KUKA KRL program: MyProgram_214().src

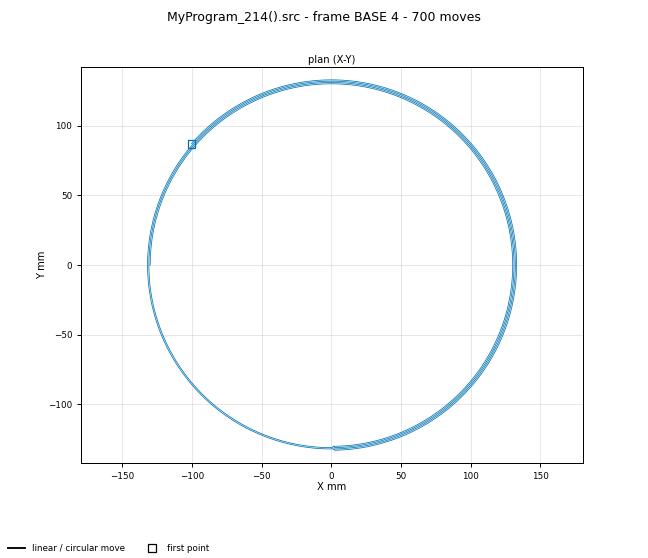
[picture p0: tool path of MyProgram_214().src in frame BASE 4, 700 of 700 moves have a stored position in this frame; points joined in program order, loops and branches not executed]
&ACCESS RVP
&REL 1
&PARAM TEMPLATE = C:\KRC\Roboter\Template\vorgabe
&PARAM EDITMASK = *
DEF MyProgram_214()
; ---- Setting reference (Base) ----
$BASE = BASE_DATA[4]

; --------------------------
; ---- Setting tool (TCP) ----
$TOOL = TOOL_DATA[3]
; --------------------------

$VEL.CP = VEL_APROX_PRINT
Startdeposition()
$VEL.CP = VEL_PRINT
LIN {X -100.4388,Y 87.0918,Z 151,A 134.8653,B 24.9546,C -1.5571,E1 24.88,E2 311.6569} C_DIS
LIN {X -97.4853,Y 90.385,Z 151,A 132.6847,B 24.9551,C -1.5488,E1 24.8842,E2 313.8668} C_DIS
LIN {X -94.8975,Y 93.098,Z 151,A 131.7947,B 24.9528,C -1.588,E1 24.8858,E2 314.6673} C_DIS
LIN {X -91.5567,Y 96.3862,Z 151,A 129.3125,B 24.9538,C -1.5705,E1 24.8908,E2 317.2017} C_DIS
LIN {X -88.2855,Y 99.3908,Z 151,A 127.4483,B 24.9534,C -1.5774,E1 24.8947,E2 319.0568} C_DIS
LIN {X -85.0766,Y 102.1512,Z 151,A 125.5893,B 24.9532,C -1.5799,E1 24.8986,E2 320.9171} C_DIS
LIN {X -81.7688,Y 104.8179,Z 151,A 123.7103,B 24.9532,C -1.5816,E1 24.9027,E2 322.799} C_DIS
LIN {X -78.285,Y 107.4446,Z 151,A 121.8187,B 24.9529,C -1.5851,E1 24.907,E2 324.689} C_DIS
LIN {X -73.7365,Y 110.6151,Z 151,A 119.6758,B 24.9519,C -1.602,E1 24.9118,E2 326.7989} C_DIS
LIN {X -71.2777,Y 112.2158,Z 151,A 117.1039,B 24.9555,C -1.5409,E1 24.9183,E2 329.5241} C_DIS
LIN {X -64.6233,Y 116.1752,Z 151,A 114.9748,B 24.9517,C -1.6057,E1 24.9231,E2 331.5056} C_DIS
LIN {X -61.5732,Y 117.8179,Z 151,A 113.4543,B 24.9517,C -1.6069,E1 24.9268,E2 333.0274} C_DIS
LIN {X -58.7566,Y 119.2473,Z 151,A 112.0651,B 24.9516,C -1.6078,E1 24.9303,E2 334.4182} C_DIS
LIN {X -55.4133,Y 120.8379,Z 151,A 110.1509,B 24.9524,C -1.5946,E1 24.9353,E2 336.3686} C_DIS
LIN {X -52.4162,Y 122.1677,Z 151,A 108.9463,B 24.9516,C -1.607,E1 24.9383,E2 337.5466} C_DIS
LIN {X -47.8757,Y 124.0173,Z 151,A 106.9413,B 24.9511,C -1.6153,E1 24.9434,E2 339.5362} C_DIS
LIN {X -44.7871,Y 125.1659,Z 151,A 105.4698,B 24.9511,C -1.6146,E1 24.9473,E2 341.0123} C_DIS
LIN {X -40.6937,Y 126.5558,Z 151,A 103.6048,B 24.9511,C -1.6168,E1 24.9522,E2 342.8756} C_DIS
LIN {X -37.2719,Y 127.6053,Z 151,A 102.1118,B 24.9508,C -1.6211,E1 24.9562,E2 344.361} C_DIS
LIN {X -33.9922,Y 128.5181,Z 151,A 100.6388,B 24.9507,C -1.6223,E1 24.9602,E2 345.8332} C_DIS
LIN {X -30.7948,Y 129.3218,Z 151,A 99.1974,B 24.9507,C -1.6227,E1 24.9641,E2 347.2758} C_DIS
LIN {X -27.1322,Y 130.1406,Z 151,A 97.4525,B 24.951,C -1.6177,E1 24.9689,E2 349.0346} C_DIS
LIN {X -23.3776,Y 130.8657,Z 151,A 95.9,B 24.9506,C -1.6239,E1 24.9731,E2 350.5742} C_DIS
LIN {X -19.5139,Y 131.4993,Z 151,A 94.2775,B 24.9503,C -1.6283,E1 24.9776,E2 352.1877} C_DIS
LIN {X -16.3255,Y 131.9325,Z 151,A 92.7599,B 24.9507,C -1.6226,E1 24.9818,E2 353.7199} C_DIS
LIN {X -12.6366,Y 132.3355,Z 151,A 91.2278,B 24.9504,C -1.6268,E1 24.986,E2 355.2429} C_DIS
LIN {X -8.7959,Y 132.6477,Z 151,A 89.4865,B 24.9506,C -1.6235,E1 24.9909,E2 356.9929} C_DIS
LIN {X -4.8875,Y 132.848,Z 151,A 87.7934,B 24.9506,C -1.6237,E1 24.9956,E2 358.6856} C_DIS
LIN {X -0.7243,Y 132.9356,Z 151,A 86.0869,B 24.9503,C -1.6287,E1 25.0004,E2 360.3806} C_DIS
LIN {X 3.3562,Y 132.8956,Z 151,A 84.2686,B 24.9505,C -1.6259,E1 25.0055,E2 362.2052} C_DIS
LIN {X 7.0592,Y 132.7505,Z 151,A 82.6113,B 24.9507,C -1.6229,E1 25.0101,E2 363.8691} C_DIS
LIN {X 11.1623,Y 132.468,Z 151,A 80.939,B 24.9503,C -1.6279,E1 25.0147,E2 365.5287} C_DIS
LIN {X 15.2217,Y 132.0641,Z 151,A 79.1094,B 24.9506,C -1.624,E1 25.0198,E2 367.3664} C_DIS
LIN {X 19.1309,Y 131.554,Z 151,A 77.4646,B 24.9504,C -1.6263,E1 25.0244,E2 369.0042} C_DIS
LIN {X 23.2351,Y 130.8912,Z 151,A 75.6881,B 24.9504,C -1.6265,E1 25.0292,E2 370.7785} C_DIS
LIN {X 26.6038,Y 130.2481,Z 151,A 74.2391,B 24.9504,C -1.6273,E1 25.0332,E2 372.2237} C_DIS
LIN {X 29.9615,Y 129.5174,Z 151,A 72.7953,B 24.9504,C -1.6285,E1 25.0371,E2 373.6629} C_DIS
LIN {X 33.2513,Y 128.7128,Z 151,A 71.0673,B 24.9512,C -1.6137,E1 25.0419,E2 375.4233} C_DIS
LIN {X 37.3957,Y 127.569,Z 151,A 69.4626,B 24.9505,C -1.6252,E1 25.0461,E2 376.9979} C_DIS
LIN {X 40.504,Y 126.6164,Z 151,A 68.0358,B 24.9507,C -1.6228,E1 25.0499,E2 378.4279} C_DIS
LIN {X 43.8865,Y 125.4846,Z 151,A 66.5342,B 24.9507,C -1.6233,E1 25.0539,E2 379.9254} C_DIS
LIN {X 47.0171,Y 124.3456,Z 151,A 65.071,B 24.9507,C -1.6205,E1 25.0577,E2 381.3922} C_DIS
LIN {X 49.9731,Y 123.187,Z 151,A 63.7361,B 24.9507,C -1.6208,E1 25.0612,E2 382.7233} C_DIS
LIN {X 53.173,Y 121.8405,Z 151,A 62.1619,B 24.9511,C -1.615,E1 25.0652,E2 384.3074} C_DIS
LIN {X 57.0541,Y 120.0715,Z 151,A 60.3594,B 24.9511,C -1.6147,E1 25.0698,E2 386.1061} C_DIS
LIN {X 60.1883,Y 118.5311,Z 151,A 58.8644,B 24.9512,C -1.6133,E1 25.0735,E2 387.6004} C_DIS
LIN {X 63.3667,Y 116.8655,Z 151,A 57.2441,B 24.9516,C -1.6072,E1 25.0776,E2 389.2304} C_DIS
LIN {X 67.1187,Y 114.7515,Z 151,A 55.3816,B 24.9518,C -1.6041,E1 25.0821,E2 391.0946} C_DIS
LIN {X 70.9545,Y 112.4198,Z 151,A 53.4788,B 24.9518,C -1.6028,E1 25.0866,E2 392.9946} C_DIS
LIN {X 74.748,Y 109.9344,Z 151,A 51.5216,B 24.9521,C -1.5994,E1 25.0911,E2 394.9532} C_DIS
LIN {X 78.4134,Y 107.351,Z 151,A 49.5804,B 24.9523,C -1.5955,E1 25.0955,E2 396.8967} C_DIS
LIN {X 81.9338,Y 104.6885,Z 151,A 47.6809,B 24.9525,C -1.5922,E1 25.0997,E2 398.7973} C_DIS
LIN {X 85.4737,Y 101.8185,Z 151,A 45.7486,B 24.9526,C -1.59,E1 25.1039,E2 400.7272} C_DIS
LIN {X 88.6689,Y 99.0484,Z 151,A 43.1234,B 24.9554,C -1.5437,E1 25.1096,E2 403.4512} C_DIS
LIN {X 93.3761,Y 94.6247,Z 151,A 41.4269,B 24.9523,C -1.5956,E1 25.1127,E2 405.0182} C_DIS
LIN {X 96.7972,Y 91.1213,Z 151,A 39.0631,B 24.9534,C -1.5773,E1 25.1174,E2 407.4151} C_DIS
LIN {X 99.9009,Y 87.7083,Z 151,A 37.0873,B 24.9536,C -1.5733,E1 25.1211,E2 409.3915} C_DIS
LIN {X 102.685,Y 84.4317,Z 151,A 34.7375,B 24.9554,C -1.5422,E1 25.1254,E2 411.8038} C_DIS
LIN {X 105.6622,Y 80.6739,Z 151,A 33.2496,B 24.9539,C -1.5681,E1 25.1278,E2 413.2235} C_DIS
LIN {X 108.0891,Y 77.392,Z 151,A 31.4386,B 24.9544,C -1.5608,E1 25.1308,E2 415.0431} C_DIS
LIN {X 111.4152,Y 72.522,Z 151,A 28.9273,B 24.9547,C -1.5558,E1 25.1347,E2 417.5538} C_DIS
LIN {X 113.7076,Y 68.8721,Z 151,A 27.0666,B 24.955,C -1.5506,E1 25.1374,E2 419.4172} C_DIS
LIN {X 115.9575,Y 65.0127,Z 151,A 25.1619,B 24.9552,C -1.5464,E1 25.14,E2 421.322} C_DIS
LIN {X 117.8536,Y 61.5051,Z 151,A 23.5076,B 24.9552,C -1.5451,E1 25.1422,E2 422.9707} C_DIS
LIN {X 119.3631,Y 58.5218,Z 151,A 22.1096,B 24.9554,C -1.5433,E1 25.1439,E2 424.3655} C_DIS
LIN {X 120.8024,Y 55.49,Z 151,A 20.682,B 24.9556,C -1.5401,E1 25.1456,E2 425.7928} C_DIS
LIN {X 122.0819,Y 52.6145,Z 151,A 19.3074,B 24.9558,C -1.5351,E1 25.1472,E2 427.1718} C_DIS
LIN {X 123.4807,Y 49.2446,Z 151,A 17.7585,B 24.956,C -1.5317,E1 25.1488,E2 428.7202} C_DIS
LIN {X 124.5747,Y 46.4055,Z 151,A 16.4792,B 24.9562,C -1.5295,E1 25.1501,E2 429.9975} C_DIS
LIN {X 125.6238,Y 43.485,Z 151,A 15.1246,B 24.9565,C -1.5245,E1 25.1513,E2 431.3563} C_DIS
LIN {X 126.7779,Y 39.9984,Z 151,A 13.4359,B 24.9571,C -1.5138,E1 25.1528,E2 433.0607} C_DIS
LIN {X 128.1939,Y 35.1996,Z 151,A 11.0831,B 24.9581,C -1.4963,E1 25.1546,E2 435.4412} C_DIS
LIN {X 129.0498,Y 31.92,Z 151,A 9.7239,B 24.9581,C -1.4972,E1 25.1555,E2 436.7903} C_DIS
LIN {X 130.1936,Y 26.8719,Z 151,A 7.6512,B 24.9579,C -1.4988,E1 25.1567,E2 438.8472} C_DIS
LIN {X 130.8791,Y 23.3024,Z 151,A 6.1872,B 24.9579,C -1.4994,E1 25.1575,E2 440.3012} C_DIS
LIN {X 131.4133,Y 20.074,Z 151,A 4.7537,B 24.9582,C -1.4936,E1 25.1581,E2 441.7401} C_DIS
LIN {X 131.9846,Y 15.8889,Z 151,A 2.9069,B 24.9586,C -1.4862,E1 25.1588,E2 443.5933} C_DIS
LIN {X 132.3916,Y 12.0521,Z 151,A 1.2035,B 24.959,C -1.4785,E1 25.1592,E2 445.3048} C_DIS
LIN {X 132.6954,Y 8.0211,Z 151,A -0.4485,B 24.959,C -1.4778,E1 25.1596,E2 446.9487} C_DIS
LIN {X 132.8828,Y 3.8181,Z 151,A -2.2288,B 24.9593,C -1.4736,E1 25.1597,E2 448.7283} C_DIS
LIN {X 132.9409,Y -0.0565,Z 151,A -4.036,B 24.96,C -1.4605,E1 25.1597,E2 450.5557} C_DIS
LIN {X 132.8768,Y -4.034,Z 151,A -5.6928,B 24.9602,C -1.458,E1 25.1597,E2 452.2084} C_DIS
LIN {X 132.6808,Y -8.2579,Z 151,A -7.4205,B 24.9602,C -1.4572,E1 25.1594,E2 453.9277} C_DIS
LIN {X 132.3492,Y -12.4942,Z 151,A -9.2116,B 24.9604,C -1.4534,E1 25.159,E2 455.7172} C_DIS
LIN {X 131.976,Y -15.9609,Z 151,A -10.686,B 24.9606,C -1.45,E1 25.1585,E2 457.191} C_DIS
LIN {X 131.4222,Y -20.0167,Z 151,A -12.4769,B 24.961,C -1.4426,E1 25.1578,E2 458.9885} C_DIS
LIN {X 130.8358,Y -23.5448,Z 151,A -13.9703,B 24.9611,C -1.4402,E1 25.1571,E2 460.4789} C_DIS
LIN {X 130.1488,Y -27.0919,Z 151,A -15.4977,B 24.9613,C -1.4367,E1 25.1563,E2 462.0056} C_DIS
LIN {X 129.5177,Y -29.9602,Z 151,A -16.8312,B 24.9618,C -1.4289,E1 25.1554,E2 463.3499} C_DIS
LIN {X 128.5065,Y -34.0359,Z 151,A -18.5829,B 24.9618,C -1.4262,E1 25.1542,E2 465.0979} C_DIS
LIN {X 127.5942,Y -37.3096,Z 151,A -20.0346,B 24.9621,C -1.4221,E1 25.1531,E2 466.5507} C_DIS
LIN {X 126.5809,Y -40.6152,Z 151,A -21.5149,B 24.9623,C -1.4179,E1 25.1519,E2 468.0327} C_DIS
LIN {X 125.5274,Y -43.7631,Z 151,A -22.9482,B 24.9626,C -1.4131,E1 25.1506,E2 469.469} C_DIS
LIN {X 124.3822,Y -46.9196,Z 151,A -24.3599,B 24.9627,C -1.4105,E1 25.1492,E2 470.8791} C_DIS
LIN {X 123.2285,Y -49.8703,Z 151,A -25.7499,B 24.963,C -1.4048,E1 25.1478,E2 472.2748} C_DIS
LIN {X 121.8935,Y -53.0503,Z 151,A -27.1857,B 24.9631,C -1.403,E1 25.1462,E2 473.707} C_DIS
LIN {X 120.6201,Y -55.8844,Z 151,A -28.5282,B 24.9634,C -1.3986,E1 25.1446,E2 475.0525} C_DIS
LIN {X 119.0684,Y -59.1193,Z 151,A -30.1178,B 24.9637,C -1.3915,E1 25.1427,E2 476.6505} C_DIS
LIN {X 116.2137,Y -64.5536,Z 151,A -32.5573,B 24.9636,C -1.3948,E1 25.1395,E2 479.0692} C_DIS
LIN {X 114.532,Y -67.4923,Z 151,A -34.2183,B 24.9644,C -1.3793,E1 25.1372,E2 480.7581} C_DIS
LIN {X 112.2366,Y -71.2448,Z 151,A -36.1169,B 24.9647,C -1.3736,E1 25.1343,E2 482.6606} C_DIS
LIN {X 109.8864,Y -74.819,Z 151,A -37.9465,B 24.9649,C -1.3691,E1 25.1315,E2 484.4918} C_DIS
LIN {X 107.4506,Y -78.2766,Z 151,A -39.7827,B 24.9652,C -1.3632,E1 25.1285,E2 486.333} C_DIS
LIN {X 104.7999,Y -81.7919,Z 151,A -41.6431,B 24.9654,C -1.36,E1 25.1254,E2 488.1922} C_DIS
LIN {X 102.1086,Y -85.128,Z 151,A -43.4777,B 24.9656,C -1.3557,E1 25.1221,E2 490.0284} C_DIS
LIN {X 99.3166,Y -88.3694,Z 151,A -45.3619,B 24.9659,C -1.3486,E1 25.1186,E2 491.9208} C_DIS
LIN {X 96.3224,Y -91.6235,Z 151,A -47.2304,B 24.9661,C -1.3458,E1 25.1151,E2 493.7879} C_DIS
LIN {X 93.3487,Y -94.6515,Z 151,A -49.085,B 24.9664,C -1.3398,E1 25.1114,E2 495.6487} C_DIS
LIN {X 90.095,Y -97.7531,Z 151,A -50.9585,B 24.9664,C -1.3386,E1 25.1076,E2 497.5174} C_DIS
LIN {X 86.8975,Y -100.6063,Z 151,A -52.82,B 24.9667,C -1.3334,E1 25.1037,E2 499.3837} C_DIS
LIN {X 83.421,Y -103.507,Z 151,A -54.7407,B 24.9668,C -1.3306,E1 25.0995,E2 501.3037} C_DIS
LIN {X 79.8391,Y -106.2948,Z 151,A -56.6606,B 24.967,C -1.3283,E1 25.0953,E2 503.222} C_DIS
LIN {X 76.3705,Y -108.8136,Z 151,A -58.5582,B 24.9673,C -1.3217,E1 25.0909,E2 505.1286} C_DIS
LIN {X 72.649,Y -111.3327,Z 151,A -60.4958,B 24.9675,C -1.3177,E1 25.0864,E2 507.0691} C_DIS
LIN {X 68.7594,Y -113.7757,Z 151,A -62.4257,B 24.9675,C -1.3166,E1 25.0819,E2 508.9956} C_DIS
LIN {X 65.1927,Y -115.8563,Z 151,A -64.1936,B 24.9677,C -1.3139,E1 25.0776,E2 510.7644} C_DIS
LIN {X 61.4606,Y -117.877,Z 151,A -65.9679,B 24.9677,C -1.3137,E1 25.0732,E2 512.5343} C_DIS
LIN {X 57.5779,Y -119.8212,Z 151,A -68.4329,B 24.9694,C -1.2789,E1 25.0668,E2 515.075} C_DIS
LIN {X 53.0533,Y -121.8922,Z 151,A -69.9699,B 24.968,C -1.3079,E1 25.0631,E2 516.5396} C_DIS
LIN {X 49.8357,Y -123.2424,Z 151,A -71.4774,B 24.968,C -1.3055,E1 25.0592,E2 518.0493} C_DIS
LIN {X 46.4907,Y -124.5428,Z 151,A -72.9745,B 24.968,C -1.306,E1 25.0553,E2 519.542} C_DIS
LIN {X 43.3991,Y -125.6536,Z 151,A -74.4019,B 24.9682,C -1.3035,E1 25.0515,E2 520.9724} C_DIS
LIN {X 40.152,Y -126.7289,Z 151,A -75.8395,B 24.9682,C -1.3037,E1 25.0477,E2 522.407} C_DIS
LIN {X 37.1235,Y -127.6487,Z 151,A -77.1963,B 24.9682,C -1.3025,E1 25.0441,E2 523.7643} C_DIS
LIN {X 34.004,Y -128.515,Z 151,A -78.6396,B 24.9684,C -1.2984,E1 25.0402,E2 525.2149} C_DIS
LIN {X 30.1478,Y -129.4749,Z 151,A -80.4613,B 24.9688,C -1.2909,E1 25.0352,E2 527.0517} C_DIS
LIN {X 25.2101,Y -130.5253,Z 151,A -82.5129,B 24.9686,C -1.2955,E1 25.0296,E2 529.0899} C_DIS
LIN {X 21.9398,Y -131.1144,Z 151,A -83.9404,B 24.9686,C -1.2946,E1 25.0257,E2 530.5179} C_DIS
LIN {X 18.1449,Y -131.6949,Z 151,A -85.7012,B 24.9689,C -1.2878,E1 25.0208,E2 532.2932} C_DIS
LIN {X 14.2924,Y -132.1669,Z 151,A -87.2717,B 24.9687,C -1.2922,E1 25.0164,E2 533.8522} C_DIS
LIN {X 10.5953,Y -132.5159,Z 151,A -88.9711,B 24.969,C -1.2862,E1 25.0117,E2 535.565} C_DIS
LIN {X 6.5449,Y -132.7764,Z 151,A -90.6231,B 24.9688,C -1.2906,E1 25.0071,E2 537.206} C_DIS
LIN {X 2.3712,Y -132.9165,Z 151,A -92.448,B 24.9688,C -1.2887,E1 25.002,E2 539.035} C_DIS
LIN {X 2.3712,Y -132.9165,Z 151,A -92.448,B 24.9688,C -1.2887,E1 25.002,E2 539.035} C_DIS
Enddeposition()
LIN {X 0.9367,Y -131.9874,Z 151,A -92.3022,B 23.9056,C -1.1253,E1 23.9322,E2 539.1469} C_DIS
Startdeposition()
$VEL.CP = VEL_PRINT
LIN {X 4.4041,Y -131.9216,Z 151,A -90.4423,B 23.9048,C -1.1435,E1 23.9375,E2 537.2427} C_DIS
LIN {X 7.9598,Y -131.7529,Z 151,A -88.9768,B 23.9049,C -1.1401,E1 23.9415,E2 535.786} C_DIS
LIN {X 11.3851,Y -131.5013,Z 151,A -87.4867,B 23.9049,C -1.1408,E1 23.9457,E2 534.2951} C_DIS
LIN {X 15.312,Y -131.1022,Z 151,A -85.8169,B 23.9049,C -1.1396,E1 23.9503,E2 532.6294} C_DIS
LIN {X 17.9111,Y -130.7743,Z 151,A -84.5466,B 23.9046,C -1.147,E1 23.9539,E2 531.3419} C_DIS
LIN {X 21.576,Y -130.2176,Z 151,A -83.0479,B 23.9048,C -1.1427,E1 23.958,E2 529.8556} C_DIS
LIN {X 25.5515,Y -129.4984,Z 151,A -81.1816,B 23.9045,C -1.1498,E1 23.9631,E2 527.9739} C_DIS
LIN {X 28.6235,Y -128.8542,Z 151,A -79.955,B 23.9047,C -1.1441,E1 23.9664,E2 526.763} C_DIS
LIN {X 32.1421,Y -128.0198,Z 151,A -78.3859,B 23.9047,C -1.1457,E1 23.9707,E2 525.1924} C_DIS
LIN {X 35.2215,Y -127.2071,Z 151,A -76.9633,B 23.9045,C -1.1492,E1 23.9746,E2 523.7636} C_DIS
LIN {X 37.9247,Y -126.4291,Z 151,A -75.6517,B 23.9042,C -1.1552,E1 23.9781,E2 522.4395} C_DIS
LIN {X 41.2838,Y -125.3711,Z 151,A -74.2316,B 23.9044,C -1.1515,E1 23.9818,E2 521.0313} C_DIS
LIN {X 44.4658,Y -124.2777,Z 151,A -72.7967,B 23.9044,C -1.1521,E1 23.9856,E2 519.5981} C_DIS
LIN {X 47.5366,Y -123.1357,Z 151,A -71.3914,B 23.9044,C -1.1532,E1 23.9893,E2 518.1933} C_DIS
LIN {X 50.5434,Y -121.9325,Z 151,A -69.9776,B 23.9042,C -1.1556,E1 23.9929,E2 516.7769} C_DIS
LIN {X 53.5713,Y -120.6328,Z 151,A -68.7335,B 23.9045,C -1.1482,E1 23.9961,E2 515.5541} C_DIS
LIN {X 56.1502,Y -119.4566,Z 151,A -67.3232,B 23.904,C -1.1594,E1 23.9997,E2 514.1202} C_DIS
LIN {X 59.5377,Y -117.8025,Z 151,A -65.8636,B 23.9043,C -1.153,E1 24.0033,E2 512.6804} C_DIS
LIN {X 62.3144,Y -116.3593,Z 151,A -64.234,B 23.9036,C -1.1693,E1 24.0074,E2 511.0154} C_DIS
LIN {X 66.1207,Y -114.2392,Z 151,A -62.3845,B 23.9036,C -1.1706,E1 24.0119,E2 509.1686} C_DIS
LIN {X 69.8904,Y -111.9728,Z 151,A -60.5105,B 23.9034,C -1.1724,E1 24.0164,E2 507.2965} C_DIS
LIN {X 73.137,Y -109.8797,Z 151,A -58.7744,B 23.9031,C -1.1788,E1 24.0204,E2 505.5505} C_DIS
LIN {X 76.7032,Y -107.4205,Z 151,A -56.9224,B 23.9031,C -1.1812,E1 24.0247,E2 503.6994} C_DIS
LIN {X 80.1465,Y -104.8765,Z 151,A -55.0654,B 23.9029,C -1.1851,E1 24.0288,E2 501.8398} C_DIS
LIN {X 83.6669,Y -102.0903,Z 151,A -53.1824,B 23.9029,C -1.186,E1 24.0329,E2 499.9621} C_DIS
LIN {X 86.9206,Y -99.3347,Z 151,A -51.3402,B 23.9026,C -1.1898,E1 24.0368,E2 498.1181} C_DIS
LIN {X 90.1019,Y -96.4584,Z 151,A -49.4852,B 23.9024,C -1.1939,E1 24.0406,E2 496.261} C_DIS
LIN {X 93.1608,Y -93.5073,Z 151,A -47.6528,B 23.9023,C -1.1977,E1 24.0443,E2 494.4272} C_DIS
LIN {X 96.1372,Y -90.4444,Z 151,A -45.7785,B 23.902,C -1.2034,E1 24.0479,E2 492.5473} C_DIS
LIN {X 99.0213,Y -87.2774,Z 151,A -43.95,B 23.9018,C -1.2066,E1 24.0513,E2 490.7195} C_DIS
LIN {X 101.7797,Y -84.0444,Z 151,A -42.1269,B 23.9017,C -1.2104,E1 24.0546,E2 488.8961} C_DIS
LIN {X 104.4375,Y -80.7179,Z 151,A -40.2901,B 23.9015,C -1.2148,E1 24.0578,E2 487.0576} C_DIS
LIN {X 106.9815,Y -77.3145,Z 151,A -38.4145,B 23.9011,C -1.2215,E1 24.0609,E2 485.1749} C_DIS
LIN {X 109.4085,Y -73.8399,Z 151,A -36.6302,B 23.9011,C -1.2238,E1 24.0637,E2 483.3942} C_DIS
LIN {X 111.5238,Y -70.6046,Z 151,A -34.8927,B 23.9006,C -1.2317,E1 24.0663,E2 481.6463} C_DIS
LIN {X 113.9272,Y -66.6573,Z 151,A -32.9195,B 23.9004,C -1.2358,E1 24.0692,E2 479.6736} C_DIS
LIN {X 116.0771,Y -62.8397,Z 151,A -31.1008,B 23.9004,C -1.2371,E1 24.0716,E2 477.8619} C_DIS
LIN {X 117.466,Y -60.1986,Z 151,A -29.8303,B 23.9002,C -1.2397,E1 24.0733,E2 476.5921} C_DIS
LIN {X 118.9463,Y -57.2182,Z 151,A -28.3968,B 23.9001,C -1.2435,E1 24.075,E2 475.1573} C_DIS
LIN {X 120.309,Y -54.2952,Z 151,A -26.9673,B 23.8998,C -1.2493,E1 24.0767,E2 473.7216} C_DIS
LIN {X 121.633,Y -51.2604,Z 151,A -25.5906,B 23.8998,C -1.2506,E1 24.0782,E2 472.3498} C_DIS
LIN {X 122.7662,Y -48.4872,Z 151,A -24.3318,B 23.8996,C -1.2524,E1 24.0795,E2 471.0938} C_DIS
LIN {X 123.8927,Y -45.5336,Z 151,A -22.7752,B 23.8989,C -1.2665,E1 24.081,E2 469.5117} C_DIS
LIN {X 125.1573,Y -41.9257,Z 151,A -21.3129,B 23.8992,C -1.2613,E1 24.0823,E2 468.0708} C_DIS
LIN {X 126.1136,Y -38.9557,Z 151,A -20.1173,B 23.8994,C -1.2572,E1 24.0833,E2 466.8925} C_DIS
LIN {X 126.9,Y -36.3195,Z 151,A -18.7563,B 23.8988,C -1.2698,E1 24.0844,E2 465.5087} C_DIS
LIN {X 127.8642,Y -32.7556,Z 151,A -17.1378,B 23.8985,C -1.2759,E1 24.0856,E2 463.8851} C_DIS
LIN {X 128.6037,Y -29.7204,Z 151,A -15.9959,B 23.8988,C -1.2689,E1 24.0863,E2 462.7673} C_DIS
LIN {X 129.2756,Y -26.6464,Z 151,A -14.469,B 23.8982,C -1.2818,E1 24.0872,E2 461.2179} C_DIS
LIN {X 129.9002,Y -23.4109,Z 151,A -13.0292,B 23.8979,C -1.287,E1 24.0879,E2 459.7743} C_DIS
LIN {X 130.4406,Y -20.1834,Z 151,A -11.6326,B 23.8977,C -1.2904,E1 24.0886,E2 458.3781} C_DIS
LIN {X 130.9162,Y -16.828,Z 151,A -10.036,B 23.8971,C -1.3018,E1 24.0892,E2 456.7632} C_DIS
LIN {X 131.3581,Y -12.9347,Z 151,A -8.4873,B 23.8973,C -1.2993,E1 24.0896,E2 455.2304} C_DIS
LIN {X 131.6194,Y -9.9294,Z 151,A -7.2018,B 23.8971,C -1.3023,E1 24.0899,E2 453.9454} C_DIS
LIN {X 131.8256,Y -6.6462,Z 151,A -5.7523,B 23.8968,C -1.3082,E1 24.0901,E2 452.4906} C_DIS
LIN {X 131.9626,Y -2.9298,Z 151,A -4.0166,B 23.8962,C -1.3199,E1 24.0903,E2 450.7371} C_DIS
LIN {X 131.987,Y 1.4617,Z 151,A -2.1672,B 23.896,C -1.3231,E1 24.0903,E2 448.8913} C_DIS
LIN {X 131.8992,Y 4.9799,Z 151,A -0.7407,B 23.896,C -1.3227,E1 24.0901,E2 447.4747} C_DIS
LIN {X 131.7237,Y 8.4341,Z 151,A 0.8861,B 23.8955,C -1.3343,E1 24.0899,E2 445.8297} C_DIS
LIN {X 131.3166,Y 13.3667,Z 151,A 2.9878,B 23.8952,C -1.3387,E1 24.0893,E2 443.7302} C_DIS
LIN {X 130.9162,Y 16.828,Z 151,A 4.3954,B 23.8952,C -1.338,E1 24.0888,E2 442.333} C_DIS
LIN {X 130.4742,Y 19.9665,Z 151,A 5.7706,B 23.895,C -1.3424,E1 24.0883,E2 440.9555} C_DIS
LIN {X 129.7915,Y 24.0182,Z 151,A 7.5045,B 23.8949,C -1.3454,E1 24.0874,E2 439.2249} C_DIS
LIN {X 129.0908,Y 27.5275,Z 151,A 9.027,B 23.8947,C -1.3488,E1 24.0866,E2 437.7036} C_DIS
LIN {X 128.5029,Y 30.1616,Z 151,A 10.3509,B 23.8941,C -1.3605,E1 24.0857,E2 436.359} C_DIS
LIN {X 127.6234,Y 33.6818,Z 151,A 11.8036,B 23.8941,C -1.3589,E1 24.0847,E2 434.9189} C_DIS
LIN {X 126.7707,Y 36.761,Z 151,A 12.9838,B 23.8945,C -1.3523,E1 24.0839,E2 433.7619} C_DIS
LIN {X 125.8816,Y 39.7003,Z 151,A 14.5027,B 23.8938,C -1.3662,E1 24.0826,E2 432.2182} C_DIS
LIN {X 124.8238,Y 42.9091,Z 151,A 15.9461,B 23.8936,C -1.3694,E1 24.0813,E2 430.7753} C_DIS
LIN {X 123.6986,Y 46.0519,Z 151,A 17.3645,B 23.8934,C -1.3722,E1 24.0799,E2 429.3585} C_DIS
LIN {X 122.5516,Y 49.0231,Z 151,A 18.7624,B 23.8932,C -1.3771,E1 24.0785,E2 427.9567} C_DIS
LIN {X 121.2821,Y 52.0844,Z 151,A 20.196,B 23.8929,C -1.3811,E1 24.077,E2 426.5216} C_DIS
LIN {X 119.9753,Y 55.0284,Z 151,A 21.5849,B 23.8928,C -1.3846,E1 24.0754,E2 425.1319} C_DIS
LIN {X 118.7411,Y 57.6478,Z 151,A 22.8341,B 23.8926,C -1.3878,E1 24.0738,E2 423.8821} C_DIS
LIN {X 117.1045,Y 60.9002,Z 151,A 24.47,B 23.8922,C -1.3952,E1 24.0718,E2 422.2371} C_DIS
LIN {X 114.9775,Y 64.8285,Z 151,A 26.428,B 23.8918,C -1.4015,E1 24.0691,E2 420.2743} C_DIS
LIN {X 112.7311,Y 68.6617,Z 151,A 28.3888,B 23.8914,C -1.4084,E1 24.0663,E2 418.3071} C_DIS
LIN {X 110.4793,Y 72.229,Z 151,A 30.1369,B 23.8914,C -1.4089,E1 24.0636,E2 416.567} C_DIS
LIN {X 108.1067,Y 75.7341,Z 151,A 32.0374,B 23.891,C -1.4169,E1 24.0606,E2 414.6566} C_DIS
LIN {X 105.4689,Y 79.3654,Z 151,A 33.9465,B 23.8908,C -1.4198,E1 24.0575,E2 412.7501} C_DIS
LIN {X 102.6282,Y 83.0061,Z 151,A 35.869,B 23.8908,C -1.4204,E1 24.0541,E2 410.8355} C_DIS
LIN {X 100.1318,Y 86.0011,Z 151,A 37.6253,B 23.8904,C -1.4277,E1 24.0509,E2 409.0696} C_DIS
LIN {X 97.2995,Y 89.1929,Z 151,A 39.4689,B 23.8901,C -1.4315,E1 24.0475,E2 407.2253} C_DIS
LIN {X 94.1083,Y 92.5537,Z 151,A 41.3987,B 23.8901,C -1.4318,E1 24.0438,E2 405.3037} C_DIS
LIN {X 91.0646,Y 95.55,Z 151,A 43.2439,B 23.8899,C -1.4353,E1 24.0401,E2 403.458} C_DIS
LIN {X 88.1979,Y 98.2023,Z 151,A 45.0036,B 23.8896,C -1.4421,E1 24.0364,E2 401.6889} C_DIS
LIN {X 84.7,Y 101.2348,Z 151,A 46.9819,B 23.8894,C -1.4444,E1 24.0322,E2 399.713} C_DIS
LIN {X 81.3895,Y 103.9149,Z 151,A 48.7723,B 23.8894,C -1.4449,E1 24.0283,E2 397.9284} C_DIS
LIN {X 77.9804,Y 106.4971,Z 151,A 50.6782,B 23.8891,C -1.4508,E1 24.024,E2 396.0152} C_DIS
LIN {X 74.3399,Y 109.0701,Z 151,A 52.6171,B 23.8889,C -1.4543,E1 24.0196,E2 394.0747} C_DIS
LIN {X 70.8092,Y 111.3947,Z 151,A 54.4709,B 23.8886,C -1.4582,E1 24.0152,E2 392.2177} C_DIS
LIN {X 67.2186,Y 113.5974,Z 151,A 56.2916,B 23.8885,C -1.4606,E1 24.0109,E2 390.397} C_DIS
LIN {X 63.3637,Y 115.7912,Z 151,A 58.1711,B 23.8885,C -1.461,E1 24.0063,E2 388.5223} C_DIS
LIN {X 60.1986,Y 117.466,Z 151,A 59.63,B 23.8886,C -1.4583,E1 24.0027,E2 387.0744} C_DIS
LIN {X 57.2182,Y 118.9463,Z 151,A 61.0822,B 23.8886,C -1.4605,E1 23.9991,E2 385.6207} C_DIS
LIN {X 54.2715,Y 120.3196,Z 151,A 62.317,B 23.8889,C -1.4533,E1 23.996,E2 384.407} C_DIS
LIN {X 51.6256,Y 121.4805,Z 151,A 63.8281,B 23.8881,C -1.4676,E1 23.992,E2 382.8644} C_DIS
LIN {X 48.5628,Y 122.7368,Z 151,A 65.2364,B 23.8881,C -1.4676,E1 23.9884,E2 381.4594} C_DIS
LIN {X 45.0038,Y 124.0837,Z 151,A 66.8008,B 23.8882,C -1.4649,E1 23.9843,E2 379.9053} C_DIS
LIN {X 42.0289,Y 125.1229,Z 151,A 68.1673,B 23.8882,C -1.466,E1 23.9807,E2 378.5389} C_DIS
LIN {X 38.9557,Y 126.1136,Z 151,A 69.5661,B 23.8882,C -1.467,E1 23.977,E2 377.1404} C_DIS
LIN {X 35.8894,Y 127.0203,Z 151,A 70.7763,B 23.8886,C -1.4591,E1 23.9738,E2 375.9516} C_DIS
LIN {X 33.2401,Y 127.7412,Z 151,A 72.2735,B 23.8877,C -1.4751,E1 23.9696,E2 374.4175} C_DIS
LIN {X 29.7204,Y 128.6037,Z 151,A 73.5313,B 23.8885,C -1.4604,E1 23.9663,E2 373.1979} C_DIS
LIN {X 26.6464,Y 129.2756,Z 151,A 75.1036,B 23.8879,C -1.4713,E1 23.962,E2 371.6008} C_DIS
LIN {X 23.6822,Y 129.8517,Z 151,A 76.4047,B 23.8879,C -1.4713,E1 23.9584,E2 370.3012} C_DIS
LIN {X 20.9589,Y 130.3205,Z 151,A 77.7047,B 23.8876,C -1.4767,E1 23.9548,E2 368.9893} C_DIS
LIN {X 17.2974,Y 130.8547,Z 151,A 79.1863,B 23.8879,C -1.471,E1 23.9507,E2 367.5231} C_DIS
LIN {X 14.198,Y 131.2271,Z 151,A 80.5251,B 23.8879,C -1.4704,E1 23.947,E2 366.1867} C_DIS
LIN {X 11.198,Y 131.5171,Z 151,A 81.7725,B 23.8881,C -1.4676,E1 23.9436,E2 364.9471} C_DIS
LIN {X 8.4341,Y 131.7237,Z 151,A 82.8678,B 23.8884,C -1.4624,E1 23.9406,E2 363.8653} C_DIS
LIN {X 5.4442,Y 131.8811,Z 151,A 84.3664,B 23.8878,C -1.4721,E1 23.9363,E2 362.3433} C_DIS
LIN {X 2.0893,Y 131.9766,Z 151,A 85.8568,B 23.8878,C -1.4735,E1 23.9321,E2 360.8494} C_DIS
LIN {X -2.0372,Y 131.9775,Z 151,A 87.538,B 23.8881,C -1.4678,E1 23.9275,E2 359.1824} C_DIS
LIN {X -4.9465,Y 131.9005,Z 151,A 88.8969,B 23.8878,C -1.4721,E1 23.9237,E2 357.8127} C_DIS
LIN {X -8.4341,Y 131.7237,Z 151,A 90.5328,B 23.8875,C -1.4774,E1 23.9191,E2 356.1633} C_DIS
LIN {X -12.3279,Y 131.4163,Z 151,A 92.054,B 23.8881,C -1.4681,E1 23.9149,E2 354.6641} C_DIS
LIN {X -15.312,Y 131.1022,Z 151,A 93.3721,B 23.8881,C -1.4681,E1 23.9112,E2 353.3451} C_DIS
LIN {X -17.9111,Y 130.7743,Z 151,A 94.6462,B 23.8877,C -1.474,E1 23.9077,E2 352.0554} C_DIS
LIN {X -20.9589,Y 130.3205,Z 151,A 95.9891,B 23.8877,C -1.4734,E1 23.904,E2 350.713} C_DIS
LIN {X -24.0182,Y 129.7915,Z 151,A 97.3655,B 23.8877,C -1.4737,E1 23.9002,E2 349.3341} C_DIS
LIN {X -27.5275,Y 129.0908,Z 151,A 98.5901,B 23.8887,C -1.4566,E1 23.8969,E2 348.1504} C_DIS
LIN {X -30.1616,Y 128.5029,Z 151,A 100.0787,B 23.8879,C -1.4707,E1 23.8928,E2 346.6248} C_DIS
LIN {X -33.6818,Y 127.6234,Z 151,A 101.5224,B 23.8884,C -1.4629,E1 23.8889,E2 345.1983} C_DIS
LIN {X -36.9312,Y 126.7209,Z 151,A 102.9932,B 23.8884,C -1.4617,E1 23.885,E2 343.728} C_DIS
LIN {X -40.9339,Y 125.4876,Z 151,A 104.9571,B 23.8882,C -1.4665,E1 23.8797,E2 341.7485} C_DIS
LIN {X -44.4417,Y 124.2864,Z 151,A 106.4566,B 23.8886,C -1.4592,E1 23.8758,E2 340.2638} C_DIS
LIN {X -47.5765,Y 123.1202,Z 151,A 107.8995,B 23.8887,C -1.4569,E1 23.872,E2 338.8236} C_DIS
LIN {X -50.5434,Y 121.9325,Z 151,A 109.2839,B 23.8888,C -1.4548,E1 23.8685,E2 337.4412} C_DIS
LIN {X -53.5713,Y 120.6328,Z 151,A 110.5358,B 23.8894,C -1.4442,E1 23.8653,E2 336.2123} C_DIS
LIN {X -56.1502,Y 119.4566,Z 151,A 111.9562,B 23.889,C -1.4513,E1 23.8617,E2 334.7707} C_DIS
LIN {X -59.4899,Y 117.8268,Z 151,A 113.5879,B 23.8891,C -1.4496,E1 23.8576,E2 333.1387} C_DIS
LIN {X -62.8397,Y 116.0771,Z 151,A 115.3531,B 23.8889,C -1.4527,E1 23.8532,E2 331.3606} C_DIS
LIN {X -66.7018,Y 113.901,Z 151,A 117.2623,B 23.8892,C -1.4485,E1 23.8486,E2 329.4557} C_DIS
LIN {X -70.6046,Y 111.5238,Z 151,A 119.2153,B 23.8895,C -1.4434,E1 23.844,E2 327.5092} C_DIS
LIN {X -73.8399,Y 109.4085,Z 151,A 120.9426,B 23.8895,C -1.4424,E1 23.8399,E2 325.7782} C_DIS
LIN {X -77.3145,Y 106.9815,Z 151,A 122.7919,B 23.8897,C -1.4391,E1 23.8357,E2 323.9305} C_DIS
LIN {X -80.9409,Y 104.2646,Z 151,A 124.7196,B 23.8901,C -1.4331,E1 23.8315,E2 322.0103} C_DIS
LIN {X -84.0444,Y 101.7797,Z 151,A 126.5042,B 23.8901,C -1.432,E1 23.8276,E2 320.2213} C_DIS
LIN {X -87.561,Y 98.7706,Z 151,A 128.4508,B 23.8905,C -1.4245,E1 23.8235,E2 318.2853} C_DIS
LIN {X -90.6029,Y 95.9877,Z 151,A 130.2981,B 23.8906,C -1.423,E1 23.8197,E2 316.4338} C_DIS
LIN {X -93.5073,Y 93.1608,Z 151,A 132.0921,B 23.8908,C -1.4203,E1 23.8162,E2 314.6386} C_DIS
LIN {X -96.7204,Y 89.8205,Z 151,A 134.0419,B 23.8912,C -1.4124,E1 23.8125,E2 312.6994} C_DIS
LIN {X -99.4098,Y 86.8345,Z 151,A 135.8436,B 23.8913,C -1.4106,E1 23.8091,E2 310.8938} C_DIS
LIN {X -102.0903,Y 83.6669,Z 151,A 137.6801,B 23.8915,C -1.4075,E1 23.8058,E2 309.0561} C_DIS
LIN {X -104.9555,Y 80.0432,Z 151,A 139.6237,B 23.892,C -1.3992,E1 23.8025,E2 307.1233} C_DIS
LIN {X -107.4945,Y 76.5996,Z 151,A 141.4861,B 23.8922,C -1.3943,E1 23.7995,E2 305.2634} C_DIS
LIN {X -109.8797,Y 73.137,Z 151,A 143.3266,B 23.8925,C -1.3899,E1 23.7966,E2 303.4243} C_DIS
LIN {X -112.1812,Y 69.5555,Z 151,A 145.2413,B 23.8925,C -1.3877,E1 23.7937,E2 301.5049} C_DIS
LIN {X -114.4439,Y 65.767,Z 151,A 147.2081,B 23.8928,C -1.3845,E1 23.7909,E2 299.5354} C_DIS
LIN {X -116.4728,Y 62.1031,Z 151,A 149.0526,B 23.893,C -1.3803,E1 23.7885,E2 297.691} C_DIS
LIN {X -118.2163,Y 58.7116,Z 151,A 150.5725,B 23.8936,C -1.3692,E1 23.7866,E2 296.1902} C_DIS
LIN {X -119.6559,Y 55.719,Z 151,A 151.8375,B 23.8943,C -1.3567,E1 23.7851,E2 294.9489} C_DIS
LIN {X -120.8263,Y 53.1387,Z 151,A 153.3899,B 23.8937,C -1.3677,E1 23.7833,E2 293.3602} C_DIS
LIN {X -122.1605,Y 49.9935,Z 151,A 154.8467,B 23.894,C -1.3619,E1 23.7818,E2 291.9093} C_DIS
LIN {X -123.529,Y 46.5045,Z 151,A 156.31,B 23.8947,C -1.3494,E1 23.7803,E2 290.4685} C_DIS
LIN {X -124.5882,Y 43.5887,Z 151,A 157.7668,B 23.8947,C -1.3502,E1 23.7789,E2 289.001} C_DIS
LIN {X -125.6785,Y 40.3361,Z 151,A 159.195,B 23.895,C -1.3427,E1 23.7777,E2 287.5828} C_DIS
LIN {X -126.6117,Y 37.3042,Z 151,A 160.5608,B 23.8953,C -1.3378,E1 23.7766,E2 286.2209} C_DIS
LIN {X -127.3306,Y 34.7799,Z 151,A 161.7699,B 23.8953,C -1.3373,E1 23.7757,E2 285.0056} C_DIS
LIN {X -128.251,Y 31.2067,Z 151,A 163.415,B 23.8955,C -1.3342,E1 23.7746,E2 283.3582} C_DIS
LIN {X -129.2756,Y 26.6464,Z 151,A 165.4206,B 23.8959,C -1.3266,E1 23.7734,E2 281.3591} C_DIS
LIN {X -129.7915,Y 24.0182,Z 151,A 166.7247,B 23.8957,C -1.3292,E1 23.7727,E2 280.0402} C_DIS
LIN {X -130.3205,Y 20.9589,Z 151,A 168.1118,B 23.8959,C -1.3266,E1 23.7721,E2 278.6509} C_DIS
LIN {X -130.7743,Y 17.9111,Z 151,A 169.2904,B 23.8965,C -1.315,E1 23.7716,E2 277.4938} C_DIS
LIN {X -131.2006,Y 14.4442,Z 151,A 170.8589,B 23.8965,C -1.3125,E1 23.7711,E2 275.9218} C_DIS
LIN {X -131.4733,Y 11.7171,Z 151,A 172.0957,B 23.8967,C -1.3107,E1 23.7708,E2 274.6815} C_DIS
LIN {X -131.7237,Y 8.4341,Z 151,A 173.2812,B 23.8975,C -1.2949,E1 23.7706,E2 273.5278} C_DIS
LIN {X -131.8857,Y 5.3247,Z 151,A 174.6055,B 23.8978,C -1.2892,E1 23.7704,E2 272.2091} C_DIS
LIN {X -131.9696,Y 2.5087,Z 151,A 175.8718,B 23.8978,C -1.2872,E1 23.7704,E2 270.9399} C_DIS
LIN {X -131.9946,Y -0.3989,Z 151,A 177.2332,B 23.8978,C -1.2876,E1 23.7703,E2 269.5689} C_DIS
LIN {X -131.9509,Y -3.3526,Z 151,A 178.4354,B 23.8983,C -1.2798,E1 23.7703,E2 268.3785} C_DIS
LIN {X -131.8364,Y -6.4304,Z 151,A 179.9922,B 23.898,C -1.2855,E1 23.7705,E2 266.7976} C_DIS
LIN {X -131.5517,Y -10.7894,Z 151,A -178.3052,B 23.8987,C -1.2705,E1 23.7709,E2 265.1216} C_DIS
LIN {X -131.2545,Y -13.944,Z 151,A -176.7867,B 23.8987,C -1.2726,E1 23.7713,E2 263.5882} C_DIS
LIN {X -130.9162,Y -16.828,Z 151,A -175.4398,B 23.8987,C -1.2725,E1 23.7717,E2 262.2331} C_DIS
LIN {X -130.489,Y -19.8709,Z 151,A -174.2483,B 23.8992,C -1.2617,E1 23.7722,E2 261.061} C_DIS
LIN {X -129.9869,Y -22.9264,Z 151,A -172.9495,B 23.8995,C -1.2553,E1 23.7728,E2 259.7698} C_DIS
LIN {X -129.4984,Y -25.5515,Z 151,A -171.4571,B 23.8989,C -1.267,E1 23.7736,E2 258.2393} C_DIS
LIN {X -128.7326,Y -29.1557,Z 151,A -169.9683,B 23.8994,C -1.2569,E1 23.7745,E2 256.7664} C_DIS
LIN {X -127.9835,Y -32.2854,Z 151,A -168.6052,B 23.8997,C -1.251,E1 23.7754,E2 255.4096} C_DIS
LIN {X -127.2071,Y -35.2215,Z 151,A -167.2149,B 23.8997,C -1.2502,E1 23.7764,E2 254.0127} C_DIS
LIN {X -126.3202,Y -38.2807,Z 151,A -165.8901,B 23.9001,C -1.2433,E1 23.7775,E2 252.6971} C_DIS
LIN {X -125.3122,Y -41.4604,Z 151,A -164.4257,B 23.9002,C -1.2396,E1 23.7787,E2 251.2329} C_DIS
LIN {X -124.2864,Y -44.4417,Z 151,A -163.0216,B 23.9004,C -1.2372,E1 23.78,E2 249.8266} C_DIS
LIN {X -123.1503,Y -47.4991,Z 151,A -161.5946,B 23.9005,C -1.2335,E1 23.7814,E2 248.4003} C_DIS
LIN {X -121.9325,Y -50.5434,Z 151,A -160.137,B 23.9007,C -1.2309,E1 23.783,E2 246.9406} C_DIS
LIN {X -120.6328,Y -53.5713,Z 151,A -158.9045,B 23.9013,C -1.2175,E1 23.7843,E2 245.734} C_DIS
LIN {X -119.2834,Y -56.5127,Z 151,A -157.3116,B 23.9011,C -1.2222,E1 23.7862,E2 244.1203} C_DIS
LIN {X -117.8832,Y -59.3792,Z 151,A -155.8325,B 23.9011,C -1.2227,E1 23.7881,E2 242.6317} C_DIS
LIN {X -116.0771,Y -62.8397,Z 151,A -154.0746,B 23.9011,C -1.2209,E1 23.7904,E2 240.8685} C_DIS
LIN {X -113.901,Y -66.7018,Z 151,A -152.1615,B 23.9014,C -1.2151,E1 23.7931,E2 238.9591} C_DIS
LIN {X -111.5238,Y -70.6046,Z 151,A -150.2368,B 23.9018,C -1.2071,E1 23.7959,E2 237.044} C_DIS
LIN {X -109.2519,Y -74.0714,Z 151,A -148.4116,B 23.902,C -1.2036,E1 23.7987,E2 235.2179} C_DIS
LIN {X -106.8921,Y -77.4378,Z 151,A -146.591,B 23.9021,C -1.2008,E1 23.8017,E2 233.395} C_DIS
LIN {X -104.3871,Y -80.7828,Z 151,A -144.743,B 23.9023,C -1.1979,E1 23.8048,E2 231.5448} C_DIS
LIN {X -101.5443,Y -84.3287,Z 151,A -142.7893,B 23.9025,C -1.1923,E1 23.8082,E2 229.5955} C_DIS
LIN {X -98.7387,Y -87.5972,Z 151,A -140.8869,B 23.9026,C -1.1895,E1 23.8117,E2 227.691} C_DIS
LIN {X -95.7193,Y -90.8875,Z 151,A -138.8953,B 23.9027,C -1.1877,E1 23.8155,E2 225.6948} C_DIS
LIN {X -92.7286,Y -93.9368,Z 151,A -137.0317,B 23.9029,C -1.1841,E1 23.8192,E2 223.8317} C_DIS
LIN {X -89.6412,Y -96.8874,Z 151,A -135.1714,B 23.9031,C -1.1806,E1 23.823,E2 221.9722} C_DIS
LIN {X -86.3776,Y -99.8075,Z 151,A -133.2671,B 23.9032,C -1.177,E1 23.827,E2 220.0689} C_DIS
LIN {X -83.0061,Y -102.6282,Z 151,A -131.3708,B 23.9034,C -1.1728,E1 23.8311,E2 218.1755} C_DIS
LIN {X -79.3654,Y -105.4689,Z 151,A -129.4319,B 23.9037,C -1.166,E1 23.8354,E2 216.246} C_DIS
LIN {X -76.2283,Y -107.7581,Z 151,A -127.6681,B 23.9037,C -1.1668,E1 23.8394,E2 214.4737} C_DIS
LIN {X -72.4212,Y -110.3528,Z 151,A -125.6748,B 23.9039,C -1.1632,E1 23.844,E2 212.4824} C_DIS
LIN {X -68.6617,Y -112.7311,Z 151,A -123.7018,B 23.9039,C -1.1623,E1 23.8487,E2 210.5051} C_DIS
LIN {X -64.8285,Y -114.9775,Z 151,A -121.7935,B 23.9041,C -1.1585,E1 23.8533,E2 208.6003} C_DIS
LIN {X -61.6791,Y -116.6955,Z 151,A -120.3366,B 23.9044,C -1.1516,E1 23.8569,E2 207.1562} C_DIS
LIN {X -58.6088,Y -118.267,Z 151,A -118.8672,B 23.9045,C -1.1484,E1 23.8605,E2 205.6907} C_DIS
LIN {X -55.719,Y -119.6559,Z 151,A -117.6261,B 23.9049,C -1.1394,E1 23.8636,E2 204.4685} C_DIS
LIN {X -52.9089,Y -120.9256,Z 151,A -116.1228,B 23.9047,C -1.1458,E1 23.8675,E2 202.9453} C_DIS
LIN {X -49.6003,Y -122.3189,Z 151,A -114.575,B 23.9047,C -1.1437,E1 23.8715,E2 201.3991} C_DIS
LIN {X -46.6985,Y -123.4564,Z 151,A -113.2254,B 23.9048,C -1.1422,E1 23.875,E2 200.0502} C_DIS
LIN {X -43.4608,Y -124.6326,Z 151,A -111.7201,B 23.9048,C -1.1414,E1 23.8789,E2 198.5439} C_DIS
LIN {X -40.4752,Y -125.6341,Z 151,A -110.3288,B 23.9048,C -1.1414,E1 23.8826,E2 197.1497} C_DIS
LIN {X -37.8587,Y -126.4493,Z 151,A -109.1329,B 23.9048,C -1.1409,E1 23.8858,E2 195.9531} C_DIS
LIN {X -34.7799,Y -127.3306,Z 151,A -107.743,B 23.9049,C -1.1399,E1 23.8896,E2 194.5632} C_DIS
LIN {X -31.2591,Y -128.2383,Z 151,A -106.1655,B 23.9049,C -1.139,E1 23.8938,E2 192.9857} C_DIS
LIN {X -28.018,Y -128.9849,Z 151,A -104.7543,B 23.9051,C -1.1367,E1 23.8977,E2 191.5783} C_DIS
LIN {X -25.1117,Y -129.5825,Z 151,A -103.6077,B 23.9054,C -1.1292,E1 23.9008,E2 190.4489} C_DIS
LIN {X -22.0489,Y -130.1387,Z 151,A -102.0568,B 23.905,C -1.1386,E1 23.9051,E2 188.8732} C_DIS
LIN {X -18.7388,Y -130.656,Z 151,A -100.6082,B 23.905,C -1.1379,E1 23.9091,E2 187.4249} C_DIS
LIN {X -15.312,Y -131.1022,Z 151,A -99.0391,B 23.9049,C -1.1411,E1 23.9135,E2 185.8469} C_DIS
LIN {X -11.8603,Y -131.4612,Z 151,A -97.5007,B 23.9049,C -1.1425,E1 23.9178,E2 184.3041} C_DIS
LIN {X -8.4341,Y -131.7237,Z 151,A -96.0838,B 23.9049,C -1.1388,E1 23.9217,E2 182.8958} C_DIS
LIN {X -4.9783,Y -131.8992,Z 151,A -94.5713,B 23.9049,C -1.1394,E1 23.9259,E2 181.3814} C_DIS
LIN {X 0,Y -131.9951,Z 151,A -92.3458,B 23.9048,C -1.143,E1 23.9322,E2 179.1469} C_DIS
LIN {X 0,Y -131.9951,Z 151,A -92.3458,B 23.9048,C -1.143,E1 23.9322,E2 179.1469} C_DIS
Enddeposition()
LIN {X 0.9375,Y -131.0445,Z 151,A -92.4391,B 22.8257,C -0.9274,E1 22.8438,E2 179.6503} C_DIS
Startdeposition()
$VEL.CP = VEL_PRINT
LIN {X -3.5036,Y -131.0018,Z 151,A -94.3186,B 22.8257,C -0.93,E1 22.8385,E2 181.5233} C_DIS
LIN {X -7.4624,Y -130.8372,Z 151,A -95.935,B 22.8254,C -0.9353,E1 22.8341,E2 183.1265} C_DIS
LIN {X -10.4413,Y -130.6332,Z 151,A -97.2575,B 22.8254,C -0.9345,E1 22.8304,E2 184.4515} C_DIS
LIN {X -14.0931,Y -130.2885,Z 151,A -98.9617,B 22.8256,C -0.93,E1 22.8256,E2 186.1684} C_DIS
LIN {X -18.1392,Y -129.7876,Z 151,A -100.7482,B 22.8256,C -0.9302,E1 22.8207,E2 187.9558} C_DIS
LIN {X -21.576,Y -129.26,Z 151,A -102.1378,B 22.8253,C -0.9367,E1 22.8169,E2 189.3301} C_DIS
LIN {X -23.9998,Y -128.8334,Z 151,A -103.6,B 22.826,C -0.9193,E1 22.8127,E2 190.8389} C_DIS
LIN {X -28.9062,Y -127.8208,Z 151,A -105.5176,B 22.8255,C -0.9329,E1 22.8076,E2 192.724} C_DIS
LIN {X -33.4186,Y -126.7161,Z 151,A -107.5572,B 22.8255,C -0.9336,E1 22.8021,E2 194.7648} C_DIS
LIN {X -36.2814,Y -125.927,Z 151,A -108.9292,B 22.8255,C -0.9311,E1 22.7983,E2 196.1457} C_DIS
LIN {X -39.7283,Y -124.8812,Z 151,A -110.4216,B 22.8254,C -0.9361,E1 22.7944,E2 197.6281} C_DIS
LIN {X -42.9463,Y -123.8113,Z 151,A -111.9131,B 22.8254,C -0.9369,E1 22.7904,E2 199.1206} C_DIS
LIN {X -46.0619,Y -122.6863,Z 151,A -113.3861,B 22.8254,C -0.9371,E1 22.7866,E2 200.5964} C_DIS
LIN {X -49.4737,Y -121.3516,Z 151,A -115.1031,B 22.8254,C -0.9335,E1 22.7821,E2 202.327} C_DIS
LIN {X -53.0301,Y -119.8402,Z 151,A -116.6494,B 22.8251,C -0.9418,E1 22.7782,E2 203.8558} C_DIS
LIN {X -56.4823,Y -118.2512,Z 151,A -118.3197,B 22.8251,C -0.9434,E1 22.7739,E2 205.5267} C_DIS
LIN {X -59.506,Y -116.7588,Z 151,A -119.9391,B 22.8253,C -0.9387,E1 22.7699,E2 207.1629} C_DIS
LIN {X -64.4518,Y -114.1058,Z 151,A -122.3812,B 22.8251,C -0.9426,E1 22.7639,E2 209.6028} C_DIS
LIN {X -68.2431,Y -111.8798,Z 151,A -124.316,B 22.8251,C -0.9448,E1 22.7592,E2 211.5382} C_DIS
LIN {X -70.6468,Y -110.3772,Z 151,A -125.7172,B 22.8252,C -0.9396,E1 22.7559,E2 212.9581} C_DIS
LIN {X -74.3819,Y -107.8958,Z 151,A -128.0918,B 22.8258,C -0.9245,E1 22.7503,E2 215.3806} C_DIS
LIN {X -78.5841,Y -104.8751,Z 151,A -129.8145,B 22.8247,C -0.9523,E1 22.7466,E2 217.0381} C_DIS
LIN {X -82.1254,Y -102.1251,Z 151,A -131.7497,B 22.8245,C -0.957,E1 22.7424,E2 218.9691} C_DIS
LIN {X -85.5404,Y -99.2821,Z 151,A -133.6798,B 22.8244,C -0.9613,E1 22.7383,E2 220.8963} C_DIS
LIN {X -88.8911,Y -96.294,Z 151,A -135.396,B 22.8238,C -0.9761,E1 22.7348,E2 222.5817} C_DIS
LIN {X -91.3262,Y -93.9876,Z 151,A -137.0751,B 22.824,C -0.9698,E1 22.7313,E2 224.2849} C_DIS
LIN {X -94.2769,Y -91.0274,Z 151,A -138.9538,B 22.824,C -0.9715,E1 22.7276,E2 226.1681} C_DIS
LIN {X -97.3277,Y -87.7586,Z 151,A -140.9989,B 22.824,C -0.9719,E1 22.7238,E2 228.2222} C_DIS
LIN {X -100.3117,Y -84.3307,Z 151,A -142.9491,B 22.8237,C -0.9781,E1 22.7202,E2 230.166} C_DIS
LIN {X -103.2115,Y -80.756,Z 151,A -144.9405,B 22.8235,C -0.9838,E1 22.7168,E2 232.1529} C_DIS
LIN {X -105.8,Y -77.334,Z 151,A -146.8398,B 22.8233,C -0.9875,E1 22.7136,E2 234.0529} C_DIS
LIN {X -108.221,Y -73.9081,Z 151,A -148.6884,B 22.8232,C -0.9915,E1 22.7107,E2 235.9012} C_DIS
LIN {X -110.07,Y -71.125,Z 151,A -150.3855,B 22.8234,C -0.985,E1 22.708,E2 237.6245} C_DIS
LIN {X -111.8098,Y -68.3571,Z 151,A -152.7849,B 22.8249,C -0.9474,E1 22.7045,E2 240.1351} C_DIS
LIN {X -115.825,Y -61.3053,Z 151,A -155.1088,B 22.8224,C -1.0094,E1 22.7015,E2 242.3119} C_DIS
LIN {X -117.4387,Y -58.153,Z 151,A -156.6354,B 22.8222,C -1.0147,E1 22.6996,E2 243.834} C_DIS
LIN {X -118.8163,Y -55.2844,Z 151,A -158.1139,B 22.8222,C -1.0148,E1 22.6978,E2 245.3209} C_DIS
LIN {X -120.3058,Y -51.9625,Z 151,A -159.5032,B 22.8216,C -1.0281,E1 22.6963,E2 246.6841} C_DIS
LIN {X -121.9487,Y -47.9833,Z 151,A -161.5885,B 22.8218,C -1.0249,E1 22.6941,E2 248.7908} C_DIS
LIN {X -123.1613,Y -44.7776,Z 151,A -162.8606,B 22.8212,C -1.039,E1 22.6929,E2 250.0341} C_DIS
LIN {X -124.4475,Y -41.0679,Z 151,A -164.8732,B 22.8215,C -1.0314,E1 22.691,E2 252.0792} C_DIS
LIN {X -125.6973,Y -37.066,Z 151,A -166.6256,B 22.8211,C -1.0404,E1 22.6896,E2 253.8194} C_DIS
LIN {X -126.5952,Y -33.8717,Z 151,A -168.058,B 22.8209,C -1.0457,E1 22.6886,E2 255.2474} C_DIS
LIN {X -127.3942,Y -30.7306,Z 151,A -169.5276,B 22.8208,C -1.0478,E1 22.6876,E2 256.721} C_DIS
LIN {X -128.2558,Y -26.9196,Z 151,A -171.3284,B 22.8208,C -1.0491,E1 22.6865,E2 258.5301} C_DIS
LIN {X -129.0137,Y -23.0031,Z 151,A -173.0412,B 22.8204,C -1.056,E1 22.6856,E2 260.2364} C_DIS
LIN {X -129.7044,Y -18.7209,Z 151,A -175.4155,B 22.821,C -1.0417,E1 22.6846,E2 262.6635} C_DIS
LIN {X -130.2548,Y -14.4057,Z 151,A -177.5964,B 22.8213,C -1.036,E1 22.684,E2 264.8736} C_DIS
LIN {X -130.7603,Y -8.7121,Z 151,A -179.2562,B 22.8194,C -1.0794,E1 22.6836,E2 266.4316} C_DIS
LIN {X -131.0433,Y -1.3504,Z 151,A 176.5083,B 22.8208,C -1.047,E1 22.6833,E2 270.7797} C_DIS
LIN {X -130.9565,Y 4.9154,Z 151,A 174.9203,B 22.8182,C -1.1045,E1 22.6835,E2 272.229} C_DIS
LIN {X -130.521,Y 11.7691,Z 151,A 170.754,B 22.82,C -1.0649,E1 22.6844,E2 276.5257} C_DIS
LIN {X -129.8245,Y 17.8811,Z 151,A 168.8299,B 22.8182,C -1.1058,E1 22.685,E2 278.3565} C_DIS
LIN {X -129.2356,Y 21.7221,Z 151,A 166.2893,B 22.8195,C -1.0759,E1 22.6863,E2 280.9914} C_DIS
LIN {X -128.0202,Y 28.011,Z 151,A 164.2579,B 22.8177,C -1.1171,E1 22.6874,E2 282.9291} C_DIS
LIN {X -127.087,Y 31.9784,Z 151,A 162.7207,B 22.8169,C -1.1332,E1 22.6883,E2 284.4345} C_DIS
LIN {X -125.9739,Y 36.1213,Z 151,A 160.6004,B 22.8171,C -1.1287,E1 22.6899,E2 286.5802} C_DIS
LIN {X -124.9043,Y 39.6559,Z 151,A 159.0655,B 22.8167,C -1.1372,E1 22.6912,E2 288.1028} C_DIS
LIN {X -123.7815,Y 43.0322,Z 151,A 157.4977,B 22.8165,C -1.1415,E1 22.6926,E2 289.6693} C_DIS
LIN {X -122.4594,Y 46.6675,Z 151,A 155.8197,B 22.8162,C -1.1472,E1 22.6942,E2 291.3428} C_DIS
LIN {X -121.0763,Y 50.1425,Z 151,A 154.1246,B 22.8162,C -1.1497,E1 22.696,E2 293.042} C_DIS
LIN {X -119.3916,Y 54.033,Z 151,A 152.0332,B 22.8163,C -1.1452,E1 22.6984,E2 295.1579} C_DIS
LIN {X -117.332,Y 58.3694,Z 151,A 150.0407,B 22.8158,C -1.156,E1 22.7008,E2 297.1343} C_DIS
LIN {X -115.2282,Y 62.4236,Z 151,A 148.0348,B 22.8156,C -1.1614,E1 22.7034,E2 299.1379} C_DIS
LIN {X -112.9251,Y 66.4984,Z 151,A 146.018,B 22.8152,C -1.1686,E1 22.7062,E2 301.1477} C_DIS
LIN {X -111.1287,Y 69.4591,Z 151,A 144.0752,B 22.8159,C -1.1546,E1 22.7092,E2 303.1377} C_DIS
LIN {X -108.7718,Y 73.0954,Z 151,A 142.5583,B 22.8149,C -1.176,E1 22.7115,E2 304.6077} C_DIS
LIN {X -105.9016,Y 77.195,Z 151,A 140.4088,B 22.8145,C -1.1836,E1 22.7149,E2 306.749} C_DIS
LIN {X -103.3146,Y 80.6247,Z 151,A 138.4544,B 22.8145,C -1.1853,E1 22.7183,E2 308.7092} C_DIS
LIN {X -100.487,Y 84.1217,Z 151,A 136.5099,B 22.8141,C -1.1914,E1 22.7217,E2 310.6479} C_DIS
LIN {X -98.5537,Y 86.3791,Z 151,A 134.8995,B 22.8146,C -1.1814,E1 22.7247,E2 312.2924} C_DIS
LIN {X -96.0405,Y 89.1647,Z 151,A 132.9646,B 22.815,C -1.1729,E1 22.7285,E2 314.2587} C_DIS
LIN {X -92.4244,Y 92.9076,Z 151,A 131.4732,B 22.8131,C -1.212,E1 22.7312,E2 315.6557} C_DIS
LIN {X -89.0676,Y 96.1295,Z 151,A 129.1164,B 22.8135,C -1.2029,E1 22.7361,E2 318.0469} C_DIS
LIN {X -84.9846,Y 99.7575,Z 151,A 126.5564,B 22.8136,C -1.2008,E1 22.7415,E2 320.6234} C_DIS
LIN {X -82.2117,Y 102.0555,Z 151,A 125.4816,B 22.8124,C -1.2259,E1 22.7437,E2 321.6377} C_DIS
LIN {X -77.1711,Y 105.9189,Z 151,A 121.9181,B 22.8138,C -1.1975,E1 22.7519,E2 325.2888} C_DIS
LIN {X -73.1464,Y 108.7375,Z 151,A 120.2685,B 22.8125,C -1.2233,E1 22.7555,E2 326.8777} C_DIS
LIN {X -70.2436,Y 110.6347,Z 151,A 118.6757,B 22.8125,C -1.2228,E1 22.7593,E2 328.4775} C_DIS
LIN {X -66.0688,Y 113.1775,Z 151,A 116.596,B 22.8122,C -1.2292,E1 22.7642,E2 330.5477} C_DIS
LIN {X -63.047,Y 114.8881,Z 151,A 114.9598,B 22.8123,C -1.2266,E1 22.7683,E2 332.1958} C_DIS
LIN {X -58.8945,Y 117.0701,Z 151,A 113.1429,B 22.8116,C -1.2403,E1 22.7727,E2 333.9829} C_DIS
LIN {X -55.8035,Y 118.5754,Z 151,A 111.5247,B 22.8118,C -1.2375,E1 22.7768,E2 335.6127} C_DIS
LIN {X -49.7665,Y 121.2333,Z 151,A 108.5943,B 22.8117,C -1.2396,E1 22.7843,E2 338.5453} C_DIS
LIN {X -46.4335,Y 122.5471,Z 151,A 107.3026,B 22.8109,C -1.2539,E1 22.7876,E2 339.8032} C_DIS
LIN {X -39.2771,Y 125.0253,Z 151,A 103.7229,B 22.8113,C -1.2459,E1 22.7972,E2 343.4111} C_DIS
LIN {X -35.3682,Y 126.1853,Z 151,A 102.1051,B 22.8109,C -1.2551,E1 22.8014,E2 345.0079} C_DIS
LIN {X -32.0791,Y 127.0614,Z 151,A 100.5104,B 22.811,C -1.2518,E1 22.8058,E2 346.6137} C_DIS
LIN {X -27.8525,Y 128.0544,Z 151,A 98.7629,B 22.8106,C -1.2603,E1 22.8105,E2 348.3419} C_DIS
LIN {X -22.6209,Y 129.0821,Z 151,A 96.297,B 22.8108,C -1.256,E1 22.8173,E2 350.8218} C_DIS
LIN {X -18.8068,Y 129.6922,Z 151,A 94.178,B 22.8118,C -1.2378,E1 22.8233,E2 352.9897} C_DIS
LIN {X -14.7022,Y 130.2229,Z 151,A 92.7312,B 22.8109,C -1.255,E1 22.8272,E2 354.393} C_DIS
LIN {X -11.39,Y 130.5531,Z 151,A 91.4088,B 22.8105,C -1.2618,E1 22.8308,E2 355.6989} C_DIS
LIN {X -7.086,Y 130.8578,Z 151,A 89.4808,B 22.8105,C -1.2606,E1 22.8362,E2 357.6306} C_DIS
LIN {X -4.1797,Y 130.983,Z 151,A 87.9966,B 22.8111,C -1.2513,E1 22.8404,E2 359.139} C_DIS
LIN {X 0.6928,Y 131.0467,Z 151,A 86.0648,B 22.8106,C -1.2608,E1 22.8457,E2 361.0464} C_DIS
LIN {X 4.728,Y 130.9638,Z 151,A 84.2597,B 22.8106,C -1.2591,E1 22.8508,E2 362.8555} C_DIS
LIN {X 8.785,Y 130.7552,Z 151,A 82.3094,B 22.8111,C -1.251,E1 22.8563,E2 364.8256} C_DIS
LIN {X 13.7843,Y 130.3217,Z 151,A 80.3508,B 22.8105,C -1.2616,E1 22.8616,E2 366.7557} C_DIS
LIN {X 16.859,Y 129.9596,Z 151,A 78.949,B 22.8107,C -1.259,E1 22.8655,E2 368.1629} C_DIS
LIN {X 20.8456,Y 129.3814,Z 151,A 76.8794,B 22.8114,C -1.2443,E1 22.8713,E2 370.2682} C_DIS
LIN {X 24.2018,Y 128.7948,Z 151,A 75.6871,B 22.8108,C -1.2574,E1 22.8745,E2 371.4254} C_DIS
LIN {X 29.531,Y 127.6781,Z 151,A 73.2551,B 22.8109,C -1.2538,E1 22.8812,E2 373.8631} C_DIS
LIN {X 33.2132,Y 126.7708,Z 151,A 71.6236,B 22.8109,C -1.2539,E1 22.8856,E2 375.4914} C_DIS
LIN {X 36.6838,Y 125.8092,Z 151,A 70.137,B 22.8108,C -1.2569,E1 22.8895,E2 376.9676} C_DIS
LIN {X 39.7744,Y 124.8664,Z 151,A 68.7347,B 22.8108,C -1.2563,E1 22.8933,E2 378.3687} C_DIS
LIN {X 42.8897,Y 123.8309,Z 151,A 67.3071,B 22.8108,C -1.2554,E1 22.897,E2 379.7955} C_DIS
LIN {X 45.8972,Y 122.748,Z 151,A 65.8806,B 22.811,C -1.2527,E1 22.9008,E2 381.2256} C_DIS
LIN {X 49.2138,Y 121.4564,Z 151,A 64.3423,B 22.811,C -1.252,E1 22.9048,E2 382.762} C_DIS
LIN {X 51.9292,Y 120.3202,Z 151,A 62.9596,B 22.8113,C -1.246,E1 22.9084,E2 384.1563} C_DIS
LIN {X 55.9277,Y 118.516,Z 151,A 60.2922,B 22.8132,C -1.2087,E1 22.9153,E2 386.9122} C_DIS
LIN {X 61.3461,Y 115.8036,Z 151,A 58.4796,B 22.8114,C -1.2444,E1 22.9196,E2 388.6274} C_DIS
LIN {X 65.1711,Y 113.6965,Z 151,A 56.5003,B 22.8117,C -1.2383,E1 22.9244,E2 390.6158} C_DIS
LIN {X 69.6996,Y 110.9781,Z 151,A 54.1797,B 22.8119,C -1.2342,E1 22.9299,E2 392.9389} C_DIS
LIN {X 72.7362,Y 109.0116,Z 151,A 52.5329,B 22.8122,C -1.2286,E1 22.9338,E2 394.5942} C_DIS
LIN {X 76.7242,Y 106.2428,Z 151,A 50.4997,B 22.8122,C -1.2292,E1 22.9384,E2 396.618} C_DIS
LIN {X 80.4565,Y 103.4451,Z 151,A 48.4975,B 22.8123,C -1.2272,E1 22.9429,E2 398.6171} C_DIS
LIN {X 83.6729,Y 100.861,Z 151,A 46.6993,B 22.8125,C -1.2241,E1 22.9467,E2 400.4158} C_DIS
LIN {X 87.0668,Y 97.9469,Z 151,A 44.7181,B 22.8127,C -1.219,E1 22.9509,E2 402.4015} C_DIS
LIN {X 90.2651,Y 95.0076,Z 151,A 42.8132,B 22.8129,C -1.2147,E1 22.9548,E2 404.3087} C_DIS
LIN {X 93.4419,Y 91.8843,Z 151,A 40.9073,B 22.813,C -1.2126,E1 22.9586,E2 406.2112} C_DIS
LIN {X 96.5697,Y 88.5912,Z 151,A 38.9579,B 22.8132,C -1.2099,E1 22.9623,E2 408.1581} C_DIS
LIN {X 99.5277,Y 85.2552,Z 151,A 37.0458,B 22.8133,C -1.2072,E1 22.9658,E2 410.0676} C_DIS
LIN {X 102.1943,Y 82.0396,Z 151,A 35.1705,B 22.8137,C -1.2004,E1 22.9691,E2 411.9506} C_DIS
LIN {X 104.9048,Y 78.5442,Z 151,A 33.2235,B 22.8139,C -1.1951,E1 22.9724,E2 413.9011} C_DIS
LIN {X 107.5763,Y 74.8427,Z 151,A 31.151,B 22.8144,C -1.1863,E1 22.9758,E2 415.9849} C_DIS
LIN {X 110.3842,Y 70.6359,Z 151,A 29.0937,B 22.8143,C -1.188,E1 22.9789,E2 418.0264} C_DIS
LIN {X 112.6544,Y 66.956,Z 151,A 27.1062,B 22.8147,C -1.1782,E1 22.9818,E2 420.0278} C_DIS
LIN {X 115.1186,Y 62.6245,Z 151,A 25.0459,B 22.8147,C -1.1781,E1 22.9846,E2 422.0765} C_DIS
LIN {X 116.6752,Y 59.6701,Z 151,A 23.7864,B 22.8145,C -1.1839,E1 22.9862,E2 423.3138} C_DIS
LIN {X 119.127,Y 54.6126,Z 151,A 21.1064,B 22.8153,C -1.166,E1 22.9894,E2 426.0237} C_DIS
LIN {X 120.7664,Y 50.8846,Z 151,A 18.9733,B 22.8164,C -1.1435,E1 22.9918,E2 428.2014} C_DIS
LIN {X 122.3709,Y 46.8973,Z 151,A 17.47,B 22.8158,C -1.1564,E1 22.9933,E2 429.6626} C_DIS
LIN {X 123.7093,Y 43.2405,Z 151,A 15.8899,B 22.8158,C -1.1574,E1 22.9948,E2 431.2303} C_DIS
LIN {X 124.8008,Y 39.9799,Z 151,A 14.4882,B 22.8158,C -1.1579,E1 22.996,E2 432.6219} C_DIS
LIN {X 125.715,Y 37.0056,Z 151,A 13.0767,B 22.8161,C -1.1512,E1 22.9971,E2 434.0416} C_DIS
LIN {X 126.5648,Y 33.9859,Z 151,A 11.7552,B 22.8161,C -1.1495,E1 22.9981,E2 435.3592} C_DIS
LIN {X 127.9148,Y 28.495,Z 151,A 8.4705,B 22.8184,C -1.1018,E1 23.0002,E2 438.745} C_DIS
LIN {X 129.0188,Y 22.9747,Z 151,A 6.779,B 22.817,C -1.132,E1 23.001,E2 440.3483} C_DIS
LIN {X 129.6727,Y 18.9432,Z 151,A 4.9766,B 22.8173,C -1.1255,E1 23.0018,E2 442.1556} C_DIS
LIN {X 130.0683,Y 16.0053,Z 151,A 3.6055,B 22.8176,C -1.1176,E1 23.0023,E2 443.5378} C_DIS
LIN {X 130.5534,Y 11.3854,Z 151,A 1.7137,B 22.8176,C -1.118,E1 23.0028,E2 445.4162} C_DIS
LIN {X 130.8058,Y 7.9723,Z 151,A 0.2201,B 22.8178,C -1.1134,E1 23.0031,E2 446.9119} C_DIS
LIN {X 130.9857,Y 4.0839,Z 151,A -1.5122,B 22.8182,C -1.1064,E1 23.0033,E2 448.6508} C_DIS
LIN {X 131.0486,Y 0.6142,Z 151,A -3.0284,B 22.8184,C -1.1015,E1 23.0033,E2 450.1695} C_DIS
LIN {X 131.0013,Y -3.5229,Z 151,A -4.7813,B 22.8185,C -1.0984,E1 23.0033,E2 451.9186} C_DIS
LIN {X 130.8296,Y -7.5867,Z 151,A -6.6792,B 22.819,C -1.0867,E1 23.003,E2 453.8341} C_DIS
LIN {X 130.4618,Y -12.387,Z 151,A -8.6842,B 22.8191,C -1.0849,E1 23.0025,E2 455.8307} C_DIS
LIN {X 129.9638,Y -16.8266,Z 151,A -10.5633,B 22.8193,C -1.0823,E1 23.0019,E2 457.7042} C_DIS
LIN {X 129.4512,Y -20.4006,Z 151,A -12.1035,B 22.8193,C -1.0791,E1 23.0012,E2 459.2425} C_DIS
LIN {X 128.7454,Y -24.4601,Z 151,A -13.959,B 22.8198,C -1.0706,E1 23.0003,E2 461.1078} C_DIS
LIN {X 127.9806,Y -28.1946,Z 151,A -15.6695,B 22.8201,C -1.0631,E1 22.9993,E2 462.8265} C_DIS
LIN {X 127.2278,Y -31.421,Z 151,A -16.9675,B 22.82,C -1.0659,E1 22.9985,E2 464.109} C_DIS
LIN {X 124.8079,Y -39.9575,Z 151,A -20.854,B 22.8205,C -1.0532,E1 22.9955,E2 468.0033} C_DIS
LIN {X 123.5293,Y -43.7567,Z 151,A -22.5662,B 22.8207,C -1.0497,E1 22.9939,E2 469.7138} C_DIS
LIN {X 122.5976,Y -46.2986,Z 151,A -24.0951,B 22.8216,C -1.029,E1 22.9923,E2 471.2864} C_DIS
LIN {X 121.3072,Y -49.584,Z 151,A -25.4126,B 22.8213,C -1.0354,E1 22.991,E2 472.5795} C_DIS
LIN {X 119.7438,Y -53.2457,Z 151,A -27.0301,B 22.8213,C -1.0362,E1 22.9892,E2 474.1851} C_DIS
LIN {X 117.1628,Y -58.7123,Z 151,A -29.7795,B 22.8218,C -1.023,E1 22.9858,E2 476.952} C_DIS
LIN {X 115.1852,Y -62.5023,Z 151,A -31.6043,B 22.822,C -1.0197,E1 22.9834,E2 478.7747} C_DIS
LIN {X 113.45,Y -65.5987,Z 151,A -33.0952,B 22.822,C -1.0182,E1 22.9814,E2 480.261} C_DIS
LIN {X 111.461,Y -68.9251,Z 151,A -34.8456,B 22.8224,C -1.0105,E1 22.9788,E2 482.021} C_DIS
LIN {X 109.3496,Y -72.2274,Z 151,A -36.555,B 22.8226,C -1.0059,E1 22.9762,E2 483.7328} C_DIS
LIN {X 107.3396,Y -75.1829,Z 151,A -38.0965,B 22.8226,C -1.0026,E1 22.9738,E2 485.2744} C_DIS
LIN {X 104.2142,Y -79.4578,Z 151,A -40.4168,B 22.823,C -0.9961,E1 22.9699,E2 487.5992} C_DIS
LIN {X 100.4229,Y -84.1981,Z 151,A -42.9834,B 22.823,C -0.9933,E1 22.9654,E2 490.1596} C_DIS
LIN {X 97.6441,Y -87.4055,Z 151,A -44.809,B 22.8232,C -0.9901,E1 22.962,E2 491.9846} C_DIS
LIN {X 95.0628,Y -90.207,Z 151,A -46.5495,B 22.8235,C -0.9822,E1 22.9587,E2 493.7369} C_DIS
LIN {X 91.6993,Y -93.6233,Z 151,A -48.5895,B 22.8236,C -0.9798,E1 22.9546,E2 495.7733} C_DIS
LIN {X 88.5084,Y -96.6458,Z 151,A -50.4455,B 22.8236,C -0.9785,E1 22.9509,E2 497.6243} C_DIS
LIN {X 85.6085,Y -99.2234,Z 151,A -51.9393,B 22.8234,C -0.9846,E1 22.9478,E2 499.0961} C_DIS
LIN {X 83.7684,Y -100.782,Z 151,A -53.3148,B 22.8242,C -0.9665,E1 22.9448,E2 500.5121} C_DIS
LIN {X 80.0193,Y -103.784,Z 151,A -55.3572,B 22.8242,C -0.9647,E1 22.9403,E2 502.5506} C_DIS
LIN {X 76.5873,Y -106.342,Z 151,A -57.2078,B 22.8244,C -0.9618,E1 22.9361,E2 504.4014} C_DIS
LIN {X 73.9605,Y -108.185,Z 151,A -58.4207,B 22.8241,C -0.9683,E1 22.9334,E2 505.5931} C_DIS
LIN {X 70.1004,Y -110.7251,Z 151,A -60.6045,B 22.8246,C -0.9564,E1 22.9282,E2 507.7994} C_DIS
LIN {X 66.2732,Y -113.0574,Z 151,A -62.4183,B 22.8244,C -0.9598,E1 22.9239,E2 509.5982} C_DIS
LIN {X 60.679,Y -116.1538,Z 151,A -65.2828,B 22.8248,C -0.9517,E1 22.9169,E2 512.4745} C_DIS
LIN {X 56.9392,Y -118.0328,Z 151,A -66.9309,B 22.8245,C -0.9575,E1 22.9128,E2 514.1029} C_DIS
LIN {X 52.7468,Y -119.9667,Z 151,A -69.0629,B 22.8249,C -0.9488,E1 22.9073,E2 516.2511} C_DIS
LIN {X 47.7284,Y -122.0478,Z 151,A -71.4055,B 22.8249,C -0.947,E1 22.9013,E2 518.5924} C_DIS
LIN {X 44.7406,Y -123.1746,Z 151,A -72.8344,B 22.8251,C -0.9436,E1 22.8975,E2 520.0267} C_DIS
LIN {X 41.7072,Y -124.2346,Z 151,A -74.0347,B 22.8248,C -0.9517,E1 22.8944,E2 521.2037} C_DIS
LIN {X 38.5322,Y -125.2555,Z 151,A -75.7041,B 22.8252,C -0.9398,E1 22.8899,E2 522.9002} C_DIS
LIN {X 35.2615,Y -126.2151,Z 151,A -77.2136,B 22.8253,C -0.9373,E1 22.8858,E2 524.4135} C_DIS
LIN {X 31.5718,Y -127.1902,Z 151,A -78.77,B 22.8252,C -0.9409,E1 22.8816,E2 525.9579} C_DIS
LIN {X 26.2596,Y -128.3905,Z 151,A -81.2337,B 22.8254,C -0.9348,E1 22.8749,E2 528.4336} C_DIS
LIN {X 22.7389,Y -129.061,Z 151,A -82.8273,B 22.8255,C -0.9323,E1 22.8705,E2 530.0317} C_DIS
LIN {X 18.3948,Y -129.7511,Z 151,A -85.1373,B 22.8263,C -0.9128,E1 22.864,E2 532.3897} C_DIS
LIN {X 14.4808,Y -130.2465,Z 151,A -86.606,B 22.8258,C -0.9238,E1 22.86,E2 533.8288} C_DIS
LIN {X 9.8276,Y -130.6798,Z 151,A -88.5035,B 22.8256,C -0.9296,E1 22.8548,E2 535.7101} C_DIS
LIN {X 6.0817,Y -130.9082,Z 151,A -90.0706,B 22.8256,C -0.9324,E1 22.8504,E2 537.2693} C_DIS
LIN {X 2.5691,Y -131.024,Z 151,A -91.6052,B 22.8256,C -0.9321,E1 22.8461,E2 538.8045} C_DIS
LIN {X 2.5691,Y -131.024,Z 151,A -91.6052,B 22.8256,C -0.9321,E1 22.8461,E2 538.8045} C_DIS
Enddeposition()
LIN {X 0.9347,Y -130.0895,Z 151,A -91.955,B 21.8484,C -0.7903,E1 21.8628,E2 539.414} C_DIS
Startdeposition()
$VEL.CP = VEL_PRINT
LIN {X 4.4968,Y -130.0276,Z 151,A -89.5015,B 21.847,C -0.8303,E1 21.87,E2 536.8537} C_DIS
LIN {X 7.8,Y -129.8702,Z 151,A -88.635,B 21.8479,C -0.8042,E1 21.8722,E2 536.0575} C_DIS
LIN {X 11.9197,Y -129.5578,Z 151,A -86.0771,B 21.8467,C -0.8385,E1 21.8796,E2 533.4091} C_DIS
LIN {X 16.0622,Y -129.1096,Z 151,A -84.6646,B 21.8473,C -0.8204,E1 21.8833,E2 532.0467} C_DIS
LIN {X 22.3382,Y -128.1732,Z 151,A -81.8632,B 21.8473,C -0.8226,E1 21.8911,E2 529.2424} C_DIS
LIN {X 26.6201,Y -127.3528,Z 151,A -79.3348,B 21.8462,C -0.8522,E1 21.8982,E2 526.6383} C_DIS
LIN {X 31.6541,Y -126.1948,Z 151,A -77.8968,B 21.8475,C -0.8159,E1 21.9018,E2 525.3002} C_DIS
LIN {X 35.0186,Y -125.3023,Z 151,A -76.2411,B 21.8472,C -0.8231,E1 21.9063,E2 523.6282} C_DIS
LIN {X 38.244,Y -124.3559,Z 151,A -74.716,B 21.8471,C -0.8268,E1 21.9104,E2 522.0963} C_DIS
LIN {X 42.8673,Y -122.839,Z 151,A -72.5786,B 21.8471,C -0.8291,E1 21.9161,E2 519.9575} C_DIS
LIN {X 46.8702,Y -121.3681,Z 151,A -70.3509,B 21.8463,C -0.8478,E1 21.922,E2 517.6852} C_DIS
LIN {X 50.268,Y -120.0004,Z 151,A -68.8992,B 21.8465,C -0.8426,E1 21.9257,E2 516.2514} C_DIS
LIN {X 54.719,Y -118.0372,Z 151,A -67.0025,B 21.8468,C -0.8345,E1 21.9305,E2 514.3821} C_DIS
LIN {X 57.8505,Y -116.5348,Z 151,A -65.4709,B 21.8468,C -0.837,E1 21.9343,E2 512.8485} C_DIS
LIN {X 61.0036,Y -114.9166,Z 151,A -63.5318,B 21.846,C -0.8572,E1 21.9392,E2 510.8615} C_DIS
LIN {X 64.2762,Y -113.1196,Z 151,A -61.6349,B 21.8454,C -0.872,E1 21.9439,E2 508.9316} C_DIS
LIN {X 68.5754,Y -110.5662,Z 151,A -60.2001,B 21.8466,C -0.84,E1 21.9471,E2 507.5877} C_DIS
LIN {X 71.3977,Y -108.765,Z 151,A -58.3883,B 21.8459,C -0.8587,E1 21.9515,E2 505.7329} C_DIS
LIN {X 75.3112,Y -106.0933,Z 151,A -56.6989,B 21.8465,C -0.8442,E1 21.9552,E2 504.089} C_DIS
LIN {X 77.4581,Y -104.5359,Z 151,A -55.3284,B 21.846,C -0.8561,E1 21.9584,E2 502.6923} C_DIS
LIN {X 80.7438,Y -102.0196,Z 151,A -53.1061,B 21.8452,C -0.8788,E1 21.9634,E2 500.4187} C_DIS
LIN {X 83.8706,Y -99.4644,Z 151,A -51.5147,B 21.8453,C -0.8739,E1 21.9667,E2 498.8476} C_DIS
LIN {X 87.7295,Y -96.0787,Z 151,A -49.4733,B 21.8455,C -0.8687,E1 21.9709,E2 496.8296} C_DIS
LIN {X 90.8048,Y -93.1777,Z 151,A -47.2586,B 21.8447,C -0.8899,E1 21.9755,E2 494.5691} C_DIS
LIN {X 93.5664,Y -90.4034,Z 151,A -45.8098,B 21.8451,C -0.881,E1 21.9782,E2 493.1512} C_DIS
LIN {X 96.9885,Y -86.7218,Z 151,A -43.9131,B 21.8454,C -0.8715,E1 21.9817,E2 491.2896} C_DIS
LIN {X 99.2901,Y -84.0772,Z 151,A -41.6903,B 21.844,C -0.9078,E1 21.9859,E2 488.9816} C_DIS
LIN {X 102.1663,Y -80.557,Z 151,A -40.2484,B 21.8449,C -0.8863,E1 21.9883,E2 487.6049} C_DIS
LIN {X 105.9565,Y -75.503,Z 151,A -37.551,B 21.8447,C -0.8897,E1 21.9928,E2 484.9134} C_DIS
LIN {X 108.0005,Y -72.5497,Z 151,A -35.7948,B 21.8442,C -0.9024,E1 21.9956,E2 483.1334} C_DIS
LIN {X 110.1548,Y -69.2344,Z 151,A -34.1179,B 21.8442,C -0.9042,E1 21.9981,E2 481.4614} C_DIS
LIN {X 112.8763,Y -64.7027,Z 151,A -32.0409,B 21.8444,C -0.8989,E1 22.001,E2 479.411} C_DIS
LIN {X 114.4075,Y -61.9558,Z 151,A -30.3898,B 21.8437,C -0.9156,E1 22.0033,E2 477.7254} C_DIS
LIN {X 116.3615,Y -58.2018,Z 151,A -27.6098,B 21.8417,C -0.9654,E1 22.0069,E2 474.8297} C_DIS
LIN {X 119.324,Y -51.8533,Z 151,A -24.5116,B 21.8413,C -0.9753,E1 22.0103,E2 471.7246} C_DIS
LIN {X 122.0415,Y -45.0906,Z 151,A -22.8234,B 21.8439,C -0.9117,E1 22.0119,E2 470.2171} C_DIS
LIN {X 123.4242,Y -41.1511,Z 151,A -20.5455,B 21.8428,C -0.9384,E1 22.014,E2 467.8829} C_DIS
LIN {X 124.8619,Y -36.5578,Z 151,A -18.0655,B 21.8418,C -0.9624,E1 22.016,E2 465.3554} C_DIS
LIN {X 125.916,Y -32.7519,Z 151,A -16.7804,B 21.8425,C -0.9459,E1 22.0169,E2 464.1226} C_DIS
LIN {X 126.8097,Y -29.0915,Z 151,A -15.0809,B 21.8422,C -0.9531,E1 22.018,E2 462.4154} C_DIS
LIN {X 127.8375,Y -24.1794,Z 151,A -12.9995,B 21.8422,C -0.954,E1 22.0191,E2 460.3458} C_DIS
LIN {X 128.2821,Y -21.6978,Z 151,A -11.7704,B 21.8418,C -0.9632,E1 22.0197,E2 459.1005} C_DIS
LIN {X 128.8355,Y -18.125,Z 151,A -10.1743,B 21.8415,C -0.9685,E1 22.0204,E2 457.5012} C_DIS
LIN {X 129.5461,Y -12.0414,Z 151,A -7.6013,B 21.8415,C -0.9711,E1 22.0212,E2 454.9387} C_DIS
LIN {X 129.9251,Y -6.8273,Z 151,A -5.4827,B 21.8415,C -0.9697,E1 22.0216,E2 452.8385} C_DIS
LIN {X 130.0825,Y -2.3792,Z 151,A -2.9659,B 21.8401,C -1.0027,E1 22.0218,E2 450.251} C_DIS
LIN {X 130.0996,Y 1.2289,Z 151,A -1.4185,B 21.8399,C -1.0058,E1 22.0218,E2 448.7063} C_DIS
LIN {X 130.0249,Y 4.5654,Z 151,A -0.1997,B 21.8403,C -0.9984,E1 22.0216,E2 447.5155} C_DIS
LIN {X 129.8398,Y 8.2923,Z 151,A 1.4275,B 21.8401,C -1.0029,E1 22.0213,E2 445.8875} C_DIS
LIN {X 129.3131,Y 14.3289,Z 151,A 4.6494,B 21.8385,C -1.0379,E1 22.0204,E2 442.5942} C_DIS
LIN {X 128.6551,Y 19.3697,Z 151,A 6.0963,B 21.8399,C -1.0069,E1 22.0199,E2 441.24} C_DIS
LIN {X 127.7506,Y 24.6339,Z 151,A 8.9218,B 21.8386,C -1.0369,E1 22.0184,E2 438.3536} C_DIS
LIN {X 126.9947,Y 28.2814,Z 151,A 10.3539,B 21.8388,C -1.032,E1 22.0176,E2 436.9445} C_DIS
LIN {X 126.1946,Y 31.655,Z 151,A 11.7617,B 21.8388,C -1.031,E1 22.0167,E2 435.5487} C_DIS
LIN {X 125.2975,Y 35.0359,Z 151,A 13.2028,B 21.8388,C -1.031,E1 22.0156,E2 434.1174} C_DIS
LIN {X 124.4035,Y 38.0886,Z 151,A 14.5977,B 21.8387,C -1.0349,E1 22.0145,E2 432.7212} C_DIS
LIN {X 123.3749,Y 41.2995,Z 151,A 16.0777,B 21.8385,C -1.0391,E1 22.0132,E2 431.2397} C_DIS
LIN {X 122.1537,Y 44.7875,Z 151,A 17.8165,B 21.838,C -1.0491,E1 22.0115,E2 429.4853} C_DIS
LIN {X 119.0657,Y 52.4472,Z 151,A 21.2465,B 21.838,C -1.0498,E1 22.0079,E2 426.0756} C_DIS
LIN {X 117.8413,Y 55.1426,Z 151,A 22.9122,B 21.837,C -1.0706,E1 22.0059,E2 424.3647} C_DIS
LIN {X 116.4461,Y 58.0303,Z 151,A 24.0101,B 21.8375,C -1.0596,E1 22.0046,E2 423.3028} C_DIS
LIN {X 114.8027,Y 61.2205,Z 151,A 25.6998,B 21.8371,C -1.0691,E1 22.0024,E2 421.5981} C_DIS
LIN {X 112.6669,Y 65.0663,Z 151,A 27.8231,B 21.8364,C -1.0832,E1 21.9994,E2 419.4501} C_DIS
LIN {X 110.9809,Y 67.902,Z 151,A 28.8781,B 21.8371,C -1.0682,E1 21.9979,E2 418.4413} C_DIS
LIN {X 108.9764,Y 71.075,Z 151,A 31.0829,B 21.8357,C -1.0986,E1 21.9945,E2 416.1683} C_DIS
LIN {X 106.633,Y 74.5447,Z 151,A 32.4593,B 21.8365,C -1.0812,E1 21.9924,E2 414.8462} C_DIS
LIN {X 104.233,Y 77.865,Z 151,A 34.2965,B 21.8362,C -1.0872,E1 21.9893,E2 413.0032} C_DIS
LIN {X 101.577,Y 81.2998,Z 151,A 36.2387,B 21.8359,C -1.0932,E1 21.986,E2 411.0556} C_DIS
LIN {X 98.769,Y 84.6888,Z 151,A 38.1539,B 21.8358,C -1.0966,E1 21.9825,E2 409.1413} C_DIS
LIN {X 95.881,Y 87.9448,Z 151,A 40.0612,B 21.8356,C -1.1005,E1 21.979,E2 407.2335} C_DIS
LIN {X 92.7187,Y 91.2728,Z 151,A 42.0628,B 21.8354,C -1.104,E1 21.9751,E2 405.2326} C_DIS
LIN {X 89.6303,Y 94.3078,Z 151,A 43.978,B 21.8352,C -1.1084,E1 21.9712,E2 403.3149} C_DIS
LIN {X 86.4186,Y 97.2592,Z 151,A 45.9077,B 21.835,C -1.1126,E1 21.9672,E2 401.3828} C_DIS
LIN {X 82.9645,Y 100.2213,Z 151,A 47.8524,B 21.835,C -1.1138,E1 21.9631,E2 399.4438} C_DIS
LIN {X 79.6916,Y 102.843,Z 151,A 49.7004,B 21.8348,C -1.1172,E1 21.959,E2 397.5945} C_DIS
LIN {X 76.0693,Y 105.551,Z 151,A 51.7012,B 21.8346,C -1.1211,E1 21.9545,E2 395.5916} C_DIS
LIN {X 70.1403,Y 109.58,Z 151,A 55.3769,B 21.8332,C -1.1502,E1 21.9458,E2 391.8521} C_DIS
LIN {X 65.9221,Y 112.1682,Z 151,A 56.9721,B 21.8343,C -1.1265,E1 21.9421,E2 390.326} C_DIS
LIN {X 62.1166,Y 114.3198,Z 151,A 58.9257,B 21.8341,C -1.1305,E1 21.9373,E2 388.3683} C_DIS
LIN {X 58.1961,Y 116.3627,Z 151,A 61.0574,B 21.8336,C -1.1415,E1 21.932,E2 386.214} C_DIS
LIN {X 55.2533,Y 117.7901,Z 151,A 62.1543,B 21.8343,C -1.1276,E1 21.9293,E2 385.1577} C_DIS
LIN {X 52.7255,Y 118.9418,Z 151,A 63.4341,B 21.8341,C -1.1316,E1 21.926,E2 383.8709} C_DIS
LIN {X 49.5894,Y 120.2838,Z 151,A 64.9098,B 21.8341,C -1.132,E1 21.9222,E2 382.398} C_DIS
LIN {X 45.2907,Y 121.9665,Z 151,A 66.9438,B 21.834,C -1.1341,E1 21.9169,E2 380.3636} C_DIS
LIN {X 41.6376,Y 123.2623,Z 151,A 68.7359,B 21.8337,C -1.1394,E1 21.9122,E2 378.5614} C_DIS
LIN {X 38.0886,Y 124.4035,Z 151,A 70.2891,B 21.8338,C -1.1368,E1 21.9081,E2 377.0186} C_DIS
LIN {X 34.7723,Y 125.3712,Z 151,A 71.8459,B 21.8337,C -1.1395,E1 21.9039,E2 375.4577} C_DIS
LIN {X 30.7518,Y 126.4175,Z 151,A 73.6572,B 21.8337,C -1.1398,E1 21.899,E2 373.6487} C_DIS
LIN {X 26.3288,Y 127.4125,Z 151,A 75.6508,B 21.8337,C -1.1407,E1 21.8935,E2 371.6557} C_DIS
LIN {X 23.2325,Y 128.0131,Z 151,A 77.2214,B 21.8332,C -1.1493,E1 21.8892,E2 370.0639} C_DIS
LIN {X 18.6915,Y 128.7546,Z 151,A 78.8277,B 21.8341,C -1.1314,E1 21.8849,E2 368.5077} C_DIS
LIN {X 15.4818,Y 129.1795,Z 151,A 80.4767,B 21.8336,C -1.1416,E1 21.8802,E2 366.8328} C_DIS
LIN {X 11.6857,Y 129.5802,Z 151,A 82.7229,B 21.8323,C -1.1668,E1 21.8738,E2 364.5203} C_DIS
LIN {X 7.1813,Y 129.9064,Z 151,A 84.2566,B 21.8333,C -1.1467,E1 21.8697,E2 363.0413} C_DIS
LIN {X 2.5093,Y 130.0803,Z 151,A 86.2397,B 21.8335,C -1.1433,E1 21.8642,E2 361.0681} C_DIS
LIN {X -1.1634,Y 130.0997,Z 151,A 88.409,B 21.8323,C -1.1672,E1 21.8579,E2 358.8343} C_DIS
LIN {X -5.8919,Y 129.9721,Z 151,A 89.8225,B 21.8338,C -1.1372,E1 21.8542,E2 357.5012} C_DIS
LIN {X -12.5811,Y 129.4943,Z 151,A 92.8189,B 21.8338,C -1.1379,E1 21.8459,E2 354.5017} C_DIS
LIN {X -16.1919,Y 129.0942,Z 151,A 94.5118,B 21.8336,C -1.141,E1 21.8411,E2 352.799} C_DIS
LIN {X -20.483,Y 128.4827,Z 151,A 96.6136,B 21.8333,C -1.1482,E1 21.8353,E2 350.6759} C_DIS
LIN {X -26.3092,Y 127.4165,Z 151,A 98.9922,B 21.8339,C -1.1362,E1 21.8288,E2 348.3263} C_DIS
LIN {X -30.2752,Y 126.5324,Z 151,A 100.7929,B 21.8339,C -1.1352,E1 21.8239,E2 346.5258} C_DIS
LIN {X -33.6787,Y 125.6692,Z 151,A 102.3394,B 21.8339,C -1.1337,E1 21.8198,E2 344.9806} C_DIS
LIN {X -37.5393,Y 124.5716,Z 151,A 104.1899,B 21.8339,C -1.1353,E1 21.8148,E2 343.1221} C_DIS
LIN {X -44.4108,Y 122.2891,Z 151,A 107.5934,B 21.8336,C -1.1407,E1 21.8057,E2 339.6965} C_DIS
LIN {X -49.2479,Y 120.4243,Z 151,A 109.8043,B 21.8339,C -1.1345,E1 21.8,E2 337.4967} C_DIS
LIN {X -54.7348,Y 118.0299,Z 151,A 112.2431,B 21.8345,C -1.1223,E1 21.7939,E2 335.084} C_DIS
LIN {X -57.689,Y 116.6144,Z 151,A 113.6657,B 21.8347,C -1.1193,E1 21.7903,E2 333.6654} C_DIS
LIN {X -60.5111,Y 115.1752,Z 151,A 115.6204,B 21.8336,C -1.1407,E1 21.7853,E2 331.6465} C_DIS
LIN {X -64.4686,Y 113.0099,Z 151,A 117.1049,B 21.8349,C -1.116,E1 21.7819,E2 330.2237} C_DIS
LIN {X -69.9237,Y 109.7186,Z 151,A 120.0223,B 21.8349,C -1.1156,E1 21.7749,E2 327.2969} C_DIS
LIN {X -73.5269,Y 107.337,Z 151,A 122.1909,B 21.8345,C -1.1231,E1 21.7698,E2 325.0994} C_DIS
LIN {X -76.4865,Y 105.2486,Z 151,A 123.8646,B 21.8345,C -1.1232,E1 21.766,E2 323.4187} C_DIS
LIN {X -79.6539,Y 102.872,Z 151,A 125.2322,B 21.8354,C -1.1038,E1 21.7631,E2 322.0977} C_DIS
LIN {X -82.9694,Y 100.2173,Z 151,A 127.6317,B 21.8346,C -1.1219,E1 21.7578,E2 319.6387} C_DIS
LIN {X -86.5213,Y 97.168,Z 151,A 129.7218,B 21.8347,C -1.1185,E1 21.7535,E2 317.5482} C_DIS
LIN {X -89.9858,Y 93.9681,Z 151,A 131.056,B 21.8364,C -1.0827,E1 21.7509,E2 316.3042} C_DIS
LIN {X -92.1915,Y 91.8051,Z 151,A 133.082,B 21.8353,C -1.1071,E1 21.7468,E2 314.2022} C_DIS
LIN {X -95.113,Y 88.7738,Z 151,A 134.4935,B 21.8364,C -1.0842,E1 21.7442,E2 312.8457} C_DIS
LIN {X -97.8972,Y 85.6949,Z 151,A 136.3869,B 21.8364,C -1.0823,E1 21.7407,E2 310.9475} C_DIS
LIN {X -100.6971,Y 82.3865,Z 151,A 138.3323,B 21.8366,C -1.0789,E1 21.7372,E2 309.0008} C_DIS
LIN {X -103.2528,Y 79.1601,Z 151,A 140.1314,B 21.8369,C -1.0736,E1 21.7341,E2 307.2061} C_DIS
LIN {X -106.714,Y 74.4284,Z 151,A 142.6447,B 21.8373,C -1.0638,E1 21.73,E2 304.7051} C_DIS
LIN {X -108.9987,Y 71.0401,Z 151,A 144.5314,B 21.8373,C -1.0625,E1 21.7271,E2 302.811} C_DIS
LIN {X -111.0464,Y 67.7953,Z 151,A 146.4206,B 21.8373,C -1.0659,E1 21.7243,E2 300.9013} C_DIS
LIN {X -113.3196,Y 63.9229,Z 151,A 148.219,B 21.8378,C -1.0529,E1 21.7219,E2 299.1272} C_DIS
LIN {X -115.3271,Y 60.2219,Z 151,A 150.0157,B 21.8382,C -1.0452,E1 21.7195,E2 297.3402} C_DIS
LIN {X -118.6316,Y 53.4189,Z 151,A 153.1429,B 21.839,C -1.027,E1 21.7158,E2 294.2426} C_DIS
LIN {X -120.1603,Y 49.8849,Z 151,A 155.129,B 21.8387,C -1.0337,E1 21.7136,E2 292.2255} C_DIS
LIN {X -121.8676,Y 45.5549,Z 151,A 157.1271,B 21.8391,C -1.0254,E1 21.7116,E2 290.2369} C_DIS
LIN {X -122.958,Y 42.5241,Z 151,A 158.5265,B 21.8393,C -1.0203,E1 21.7103,E2 288.8421} C_DIS
LIN {X -124.0059,Y 39.3645,Z 151,A 160.0252,B 21.8394,C -1.0171,E1 21.709,E2 287.3421} C_DIS
LIN {X -125.858,Y 32.9708,Z 151,A 162.9614,B 21.8398,C -1.008,E1 21.7068,E2 284.4105} C_DIS
LIN {X -126.6543,Y 29.7697,Z 151,A 164.5844,B 21.8398,C -1.0104,E1 21.7057,E2 282.77} C_DIS
LIN {X -127.6915,Y 24.9432,Z 151,A 167.0761,B 21.8395,C -1.0166,E1 21.7043,E2 280.2446} C_DIS
LIN {X -128.3737,Y 21.1487,Z 151,A 168.1811,B 21.8408,C -0.9869,E1 21.7038,E2 279.2121} C_DIS
LIN {X -128.7856,Y 18.474,Z 151,A 169.5777,B 21.8406,C -0.9915,E1 21.7032,E2 277.7935} C_DIS
LIN {X -129.52,Y 12.3136,Z 151,A 172.1545,B 21.8412,C -0.9764,E1 21.7024,E2 275.2396} C_DIS
LIN {X -129.9498,Y 6.3359,Z 151,A 174.9653,B 21.8412,C -0.9749,E1 21.7019,E2 272.4132} C_DIS
LIN {X -130.1062,Y -0.252,Z 151,A 177.9577,B 21.8415,C -0.9692,E1 21.7018,E2 269.4152} C_DIS
Enddeposition()
END
